// TIA Portal V17 export
// export: Created 2025-04-09T08:02:46.4653844Z, ExportSetting WithDefaults, DisplayName Totally Integrated Automation Portal, DisplayVersion V17 Update 8, DisplayName TIA Portal Openness, DisplayVersion V17 Update 8, DisplayName TIA Portal Version Control Interface, DisplayVersion V17, DisplayName SINAMICS Startdrive Advanced, DisplayVersion V17 SP2, DisplayName SINAMICS Startdrive G110M, G120, G120C, G120D, G120P, G115D, DisplayVersion V17 SP2, DisplayName SINAMICS Startdrive G130, G150, S120, S150, SINAMICS MV, S210, DisplayVersion V17 SP2, DisplayName STEP 7 Professional, DisplayVersion V17 Update 8, DisplayName SINUMERIK ONE STEP 7 Toolbox, DisplayVersion V17 Update 12, DisplayName SINUMERIK ONE PLC Basic Program Plus, DisplayVersion V17 Update 12, DisplayName SINUMERIK 840D sl STEP 7 Toolbox, DisplayVersion V17 Update 12, DisplayName STEP 7 Safety, DisplayVersion V17 Update 6, DisplayName WinCC Advanced, DisplayVersion V17 Update 8
FUNCTION_BLOCK "FB1403_PROGRESSIVE_LUBRICATION_WITH_GREASE"   // FB1403, LAD
{ S7_Optimized_Access := 'FALSE' }
AUTHOR : ETXETAR
VERSION : 1.0
// stored: AutoNumber false, IsIECCheckEnabled false, SetENOAutomatically false, UDAEnableTagReadback false
   VAR_INPUT
      OPTIONS_0 : Byte := 2#0000_0000;   // OPTIONS 0
      OPTIONS_1 : Byte := 2#0000_0000;   // OPTIONS 1
      TIME_VALVE_1 : Time := T#5d;   // H=HOURS; M=MINUTES
      TIME_VALVE_2 : Time := T#5d;   // H=HOURS; M=MINUTES
      TIME_VALVE_3 : Time := T#5d;   // H=HOURS; M=MINUTES
      TIME_VALVE_4 : Time := T#5d;   // H=HOURS; M=MINUTES
      PULSES_PER_CYCLE_VALVE_1 : Int := 2;   // NUMBER OF PULSES PER CYCLE
      PULSES_PER_CYCLE_VALVE_2 : Int := 2;   // NUMBER OF PULSES PER CYCLE
      PULSES_PER_CYCLE_VALVE_3 : Int := 2;   // NUMBER OF PULSES PER CYCLE
      PULSES_PER_CYCLE_VALVE_4 : Int := 2;   // NUMBER OF PULSES PER CYCLE
      BREAKER : Bool;   // CIRCUIT BREAKER INPUT
      LOW_LEVEL_ALM : Bool;   // LOW LEVEL ALARM INPUT
      OVERPRESSURE_ALM : Bool;   // OVERPRESSURE ALARM INPUT
      LUBRICATION_DONE_1 : Bool;   // LUBRICATION_DONE 1 INPUT
      LUBRICATION_DONE_2 : Bool;   // LUBRICATION_DONE 2 INPUT
      LUBRICATION_DONE_3 : Bool;   // LUBRICATION_DONE 3 INPUT
      LUBRICATION_DONE_4 : Bool;   // LUBRICATION_DONE 4 INPUT
      LUBRICATION_DONE_5 : Bool;   // LUBRICATION_DONE 5 INPUT
      LUBRICATION_DONE_6 : Bool;   // LUBRICATION_DONE 6 INPUT
      LUBRICATION_DONE_7 : Bool;   // LUBRICATION_DONE 7 INPUT
      LUBRICATION_DONE_8 : Bool;   // LUBRICATION_DONE 8 INPUT
      LUBRICATION_DONE_9 : Bool;   // LUBRICATION_DONE 9 INPUT
      SWITCH_ON_VALVE_1_DIST_REQ_AXIS_1 : Bool;   // SWITCH ON DISTANCE REQUEST INPUT FOR VALVE 1 AXIS 1
      SWITCH_ON_VALVE_1_DIST_REQ_AXIS_2 : Bool;   // SWITCH ON DISTANCE REQUEST INPUT FOR VALVE 1 AXIS 2
      SWITCH_ON_VALVE_2_DIST_REQ_AXIS_1 : Bool;   // SWITCH ON DISTANCE REQUEST INPUT FOR VALVE 2 AXIS 1
      SWITCH_ON_VALVE_2_DIST_REQ_AXIS_2 : Bool;   // SWITCH ON DISTANCE REQUEST INPUT FOR VALVE 2 AXIS 2
      SWITCH_ON_VALVE_3_DIST_REQ : Bool;   // SWITCH ON DISTANCE REQUEST INPUT FOR VALVE 3
      SWITCH_ON_VALVE_4_DIST_REQ : Bool;   // SWITCH ON DISTANCE REQUEST INPUT FOR VALVE 4
      HMI_REQ_LINE_VALVE_1 : Bool;   // HMI REQUEST LINE
      HMI_REQ_LINE_VALVE_2 : Bool;   // HMI REQUEST LINE
      HMI_REQ_LINE_VALVE_3 : Bool;   // HMI REQUEST LINE
      HMI_REQ_LINE_VALVE_4 : Bool;   // HMI REQUEST LINE
   END_VAR
   VAR_OUTPUT
      HMI_POWER_UP_COND_OFF_VALVE_1 : Bool;   // HMI POWER UP CONDITIONS OFF
      HMI_POWER_UP_COND_ON_VALVE_1 : Bool;   // HMI POWER UP CONDITIONS ON
      HMI_POWER_UP_EXECU_LEFT_VALVE_1 : Bool;   // HMI POWER UP EXECUTABLE LEFT
      HMI_POWER_UP_EXECU_RIGHT_VALVE_1 : Bool;   // HMI POWER UP EXECUTABLE RIGHT
      HMI_POWER_UP_COND_OFF_VALVE_2 : Bool;   // HMI POWER UP CONDITIONS OFF
      HMI_POWER_UP_COND_ON_VALVE_2 : Bool;   // HMI POWER UP CONDITIONS ON
      HMI_POWER_UP_EXECU_LEFT_VALVE_2 : Bool;   // HMI POWER UP EXECUTABLE LEFT
      HMI_POWER_UP_EXECU_RIGHT_VALVE_2 : Bool;   // HMI POWER UP EXECUTABLE RIGHT
      HMI_POWER_UP_COND_OFF_VALVE_3 : Bool;   // HMI POWER UP CONDITIONS OFF
      HMI_POWER_UP_COND_ON_VALVE_3 : Bool;   // HMI POWER UP CONDITIONS ON
      HMI_POWER_UP_EXECU_LEFT_VALVE_3 : Bool;   // HMI POWER UP EXECUTABLE LEFT
      HMI_POWER_UP_EXECU_RIGHT_VALVE_3 : Bool;   // HMI POWER UP EXECUTABLE RIGHT
      HMI_POWER_UP_COND_OFF_VALVE_4 : Bool;   // HMI POWER UP CONDITIONS OFF
      HMI_POWER_UP_COND_ON_VALVE_4 : Bool;   // HMI POWER UP CONDITIONS ON
      HMI_POWER_UP_EXECU_LEFT_VALVE_4 : Bool;   // HMI POWER UP EXECUTABLE LEFT
      HMI_POWER_UP_EXECU_RIGHT_VALVE_4 : Bool;   // HMI POWER UP EXECUTABLE RIGHT
      MOTOR : Bool;   // MOTOR OUTPUT
      VALVE_1 : Bool;
      VALVE_2 : Bool;
      VALVE_3 : Bool;
      VALVE_4 : Bool;
   END_VAR
   VAR DB_SPECIFIC
      BREAKER_ALARM : Bool;   // CIRCUIT BREAKER TRIPPED ALARM
      LOW_LEVEL_ALARM : Bool;   // LOW LEVEL ALARM
      OVERPRESSURE_ALARM : Bool;   // OVERPRESSURE ALARM
      LUBRICATION_DONE_1_ALARM : Bool;   // LUBRICATION DONE 1 ALARM
      LUBRICATION_DONE_2_ALARM : Bool;   // LUBRICATION DONE 2 ALARM
      LUBRICATION_DONE_3_ALARM : Bool;   // LUBRICATION DONE 3 ALARM
      LUBRICATION_DONE_4_ALARM : Bool;   // LUBRICATION DONE 4 ALARM
      DATA_VALVE_1 : Struct
         SWITCH_ON_GENERAL_CONDITIONS : Bool;   // SWITCH ON GENERAL CONDITIONS
         SWITCH_ON_INITIAL_CONDITIONS : Bool;   // SWITCH ON INITIAL CONDITIONS
         SWITCH_ON_MANUAL_REQUEST : Bool;   // SWITCH ON MANUAL REQUEST
         SWITCH_ON_AUTO_REQUEST : Bool;   // SWITCH ON AUTO REQUEST
         SWITCH_ON_TIME_REQUEST : Bool;   // SWITCH ON TIME REQUEST
         SWITCH_ON_GLOBAL_REQUEST : Bool;   // SWITCH ON GLOBAL REQUEST
         SWITCH_ON_CMM : Bool;   // SWITCH ON COMMAND
         SWITCH_ON : Bool;   // SWITCH ON
         IN_SERVICE : Bool;   // IN SERVICE
         SWITCH_OFF_GENERAL_CONDITIONS : Bool;   // SWITCH OFF GENERAL CONDITIONS
         SWITCH_OFF_INITIAL_CONDITIONS : Bool;   // SWITCH OFF INITIAL CONDITIONS
         SWITCH_OFF_MANUAL_REQUEST : Bool;   // SWITCH OFF MANUAL REQUEST
         SWITCH_OFF_AUTO_REQUEST : Bool;   // SWITCH OFF AUTO REQUEST
         SWITCH_OFF_GLOBAL_REQUEST : Bool;   // SWITCH OFF GLOBAL REQUEST
         SWITCH_OFF_CMM : Bool;   // SWITCH OFF COMMAND
         SWITCH_OFF : Bool;   // SWITCH OFF
         OUT_OF_SERVICE : Bool;   // OUT OF SERVICE
         TIMER_1 : TON_TIME;   // TIMER_1
         PULSE_1 : Bool;   // PULSE_1
         PULSE_2 : Bool;   // PULSE_1
      END_STRUCT;
      DATA_VALVE_2 : Struct
         SWITCH_ON_GENERAL_CONDITIONS : Bool;   // SWITCH ON GENERAL CONDITIONS
         SWITCH_ON_INITIAL_CONDITIONS : Bool;   // SWITCH ON INITIAL CONDITIONS
         SWITCH_ON_MANUAL_REQUEST : Bool;   // SWITCH ON MANUAL REQUEST
         SWITCH_ON_AUTO_REQUEST : Bool;   // SWITCH ON AUTO REQUEST
         SWITCH_ON_TIME_REQUEST : Bool;   // SWITCH ON TIME REQUEST
         SWITCH_ON_GLOBAL_REQUEST : Bool;   // SWITCH ON GLOBAL REQUEST
         SWITCH_ON_CMM : Bool;   // SWITCH ON COMMAND
         SWITCH_ON : Bool;   // SWITCH ON
         IN_SERVICE : Bool;   // IN SERVICE
         SWITCH_OFF_GENERAL_CONDITIONS : Bool;   // SWITCH OFF GENERAL CONDITIONS
         SWITCH_OFF_INITIAL_CONDITIONS : Bool;   // SWITCH OFF INITIAL CONDITIONS
         SWITCH_OFF_MANUAL_REQUEST : Bool;   // SWITCH OFF MANUAL REQUEST
         SWITCH_OFF_AUTO_REQUEST : Bool;   // SWITCH OFF AUTO REQUEST
         SWITCH_OFF_GLOBAL_REQUEST : Bool;   // SWITCH OFF GLOBAL REQUEST
         SWITCH_OFF_CMM : Bool;   // SWITCH OFF COMMAND
         SWITCH_OFF : Bool;   // SWITCH OFF
         OUT_OF_SERVICE : Bool;   // OUT OF SERVICE
         TIMER_1 : TON_TIME;   // TIMER_1
         PULSE_1 : Bool;   // PULSE_1
         PULSE_2 : Bool;   // PULSE_1
      END_STRUCT;
      DATA_VALVE_3 : Struct
         SWITCH_ON_GENERAL_CONDITIONS : Bool;   // SWITCH ON GENERAL CONDITIONS
         SWITCH_ON_INITIAL_CONDITIONS : Bool;   // SWITCH ON INITIAL CONDITIONS
         SWITCH_ON_MANUAL_REQUEST : Bool;   // SWITCH ON MANUAL REQUEST
         SWITCH_ON_AUTO_REQUEST : Bool;   // SWITCH ON AUTO REQUEST
         SWITCH_ON_TIME_REQUEST : Bool;   // SWITCH ON TIME REQUEST
         SWITCH_ON_GLOBAL_REQUEST : Bool;   // SWITCH ON GLOBAL REQUEST
         SWITCH_ON_CMM : Bool;   // SWITCH ON COMMAND
         SWITCH_ON : Bool;   // SWITCH ON
         IN_SERVICE : Bool;   // IN SERVICE
         SWITCH_OFF_GENERAL_CONDITIONS : Bool;   // SWITCH OFF GENERAL CONDITIONS
         SWITCH_OFF_INITIAL_CONDITIONS : Bool;   // SWITCH OFF INITIAL CONDITIONS
         SWITCH_OFF_MANUAL_REQUEST : Bool;   // SWITCH OFF MANUAL REQUEST
         SWITCH_OFF_AUTO_REQUEST : Bool;   // SWITCH OFF AUTO REQUEST
         SWITCH_OFF_GLOBAL_REQUEST : Bool;   // SWITCH OFF GLOBAL REQUEST
         SWITCH_OFF_CMM : Bool;   // SWITCH OFF COMMAND
         SWITCH_OFF : Bool;   // SWITCH OFF
         OUT_OF_SERVICE : Bool;   // OUT OF SERVICE
         TIMER_1 : TON_TIME;   // TIMER_1
         PULSE_1 : Bool;   // PULSE_1
         PULSE_2 : Bool;   // PULSE_1
      END_STRUCT;
      DATA_VALVE_4 : Struct
         SWITCH_ON_GENERAL_CONDITIONS : Bool;   // SWITCH ON GENERAL CONDITIONS
         SWITCH_ON_INITIAL_CONDITIONS : Bool;   // SWITCH ON INITIAL CONDITIONS
         SWITCH_ON_MANUAL_REQUEST : Bool;   // SWITCH ON MANUAL REQUEST
         SWITCH_ON_AUTO_REQUEST : Bool;   // SWITCH ON AUTO REQUEST
         SWITCH_ON_TIME_REQUEST : Bool;   // SWITCH ON TIME REQUEST
         SWITCH_ON_GLOBAL_REQUEST : Bool;   // SWITCH ON GLOBAL REQUEST
         SWITCH_ON_CMM : Bool;   // SWITCH ON COMMAND
         SWITCH_ON : Bool;   // SWITCH ON
         IN_SERVICE : Bool;   // IN SERVICE
         SWITCH_OFF_GENERAL_CONDITIONS : Bool;   // SWITCH OFF GENERAL CONDITIONS
         SWITCH_OFF_INITIAL_CONDITIONS : Bool;   // SWITCH OFF INITIAL CONDITIONS
         SWITCH_OFF_MANUAL_REQUEST : Bool;   // SWITCH OFF MANUAL REQUEST
         SWITCH_OFF_AUTO_REQUEST : Bool;   // SWITCH OFF AUTO REQUEST
         SWITCH_OFF_GLOBAL_REQUEST : Bool;   // SWITCH OFF GLOBAL REQUEST
         SWITCH_OFF_CMM : Bool;   // SWITCH OFF COMMAND
         SWITCH_OFF : Bool;   // SWITCH OFF
         OUT_OF_SERVICE : Bool;   // OUT OF SERVICE
         TIMER_1 : TON_TIME;   // TIMER_1
         PULSE_1 : Bool;   // PULSE_1
         PULSE_2 : Bool;   // PULSE_1
      END_STRUCT;
      CYCLE_IN_PROCESS : Bool;   // CYCLE IN PROCESS
      ALL_LUBRICATION_DONE : Bool;   // ALL LUBRICATION DONE
      ALL_LUBRICATION_DONE_DELAYED : Bool;   // ALL LUBRICATION DONE DELAYED
      SWITCH_ON_MOTOR_REQUEST : Bool;   // SWITCH ON MOTOR REQUEST
      ANY_CYCLE_NOT_DONE : Bool;   // ANY CYCLE NOT DONE
      CYCLE_FINISHED_1 : Bool;   // CYCLE FINISHED 1
      CYCLE_FINISHED_2 : Bool;   // CYCLE FINISHED 2
      CYCLE_FINISHED_3 : Bool;   // CYCLE FINISHED 3
      CYCLE_FINISHED_4 : Bool;   // CYCLE FINISHED 4
      MANUAL_REQUEST_HELP : Bool;   // MANUAL REQUEST HELP
      SWITCH_ON_GENERAL_CONDITION_HELP : Bool;   // SWITCH ON GENERAL CONDITION HELP
      SWITCH_ON_INITIAL_CONDITION_HELP : Bool;   // SWITCH ON INITIAL CONDITION HELP
      SWITCH_OFF_GENERAL_CONDITION_HELP : Bool;   // SWITCH OFF GENERAL CONDITION HELP
      SWITCH_OFF_INITIAL_CONDITION_HELP : Bool;   // SWITCH OFF INITIAL CONDITION HELP
      ANY_ACTIVE_ALARM : Bool;   // ANY ACTIVE ALARM
      SEOC_ALARMS : Bool;   // STOP END OF CYCLE ALARMS
      WARNINGS : Bool;   // WARNINGS
      WARNINGS_GONE : Bool;   // WARNINGS GONE
      TIMER_AUX_SWTICH_ON_MOTOR : TON_TIME;   // SWTICH ON MOTOR TIMER
      TIMER_ALL_LUBRICATION_DONE : TON_TIME;   // ALL LUBRICATION DONE TIMER
      TIMER_LOW_LEVEL_ALM : TON_TIME;   // LOW LEVEL TIMER
      TIMER_OVERPRESSURE_ALM : TON_TIME;   // OVERPRESSURE TIMER
      TIMER_ANY_CYCLE_NOT_DONE : TON_TIME;   // ANY CYCLE NOT DONE TIMER
      TIMER_RUN_NIGHT_TEST : TON_TIME;   // TIMER RUN NIGHT TEST
      COUNTER_1 { S7_SetPoint := 'True'} : CTU_INT;
      COUNTER_2 { S7_SetPoint := 'True'} : CTU_INT;
      COUNTER_3 { S7_SetPoint := 'True'} : CTU_INT;
      COUNTER_4 { S7_SetPoint := 'True'} : CTU_INT;
      SEQ_GLOBAL_AUTO_REQ : Bool;   // SEQUENCE GLOBAL AUTO REQUEST
      PULSE_1 : Bool;
      PULSE_2 : Bool;
      PULSE_3 : Bool;
      PULSE_4 : Bool;
      PULSE_5 : Bool;
      PULSE_6 : Bool;
      PULSE_7 : Bool;
      PULSE_8 : Bool;
      VALVE_1_AXIS_1_DIST_MEM_REQ : Bool;   // VALVE 1 AXIS 1 DISTANCE MEMORY REQUEST
      VALVE_1_AXIS_2_DIST_MEM_REQ : Bool;   // VALVE 1 AXIS 2 DISTANCE MEMORY REQUEST
      VALVE_2_AXIS_1_DIST_MEM_REQ : Bool;   // VALVE 2 AXIS 1 DISTANCE MEMORY REQUEST
      VALVE_2_AXIS_2_DIST_MEM_REQ : Bool;   // VALVE 2 AXIS 2 DISTANCE MEMORY REQUEST
      VALVE_1_AXIS_1_2_DIST_REQ : Bool;   // VALVE 1 AXIS 1 & 2 DISTANCE REQUEST
      VALVE_2_AXIS_1_2_DIST_REQ : Bool;   // VALVE 2 AXIS 1 & 2 DISTANCE REQUEST
   END_VAR
   VAR_TEMP
      INPUTS_MASK : Byte;   // INPUT MASK
      O_BYTE_0 : Struct   // OPTIONS BYTE 0
         "CIRCUIT BREAKER" : Bool;   // CIRCUIT BREAKER OPTION
         LOW_LEVEL_ALARM : Bool;   // LOW LEVEL ALARM OPTION
         OVERPRESSURE_ALARM : Bool;   // OVERPRESSURE ALARM OPTION
         LUBRICATION_BY_TIME_VALVE_1 : Bool;   // LUBRICATE BY TIMER OR BY AUTO REQUEST OPTION
         LUBRICATION_BY_TIME_VALVE_2 : Bool;   // LUBRICATE BY TIMER OR BY AUTO REQUEST OPTION
         LUBRICATION_BY_TIME_VALVE_3 : Bool;   // LUBRICATE BY TIMER OR BY AUTO REQUEST OPTION
         LUBRICATION_BY_TIME_VALVE_4 : Bool;   // LUBRICATE BY TIMER OR BY AUTO REQUEST OPTION
         LUBRICATION_DONE_1 : Bool;   // LUBRICATION DONE 1 OPTION
      END_STRUCT;
      O_BYTE_1 : Struct   // OPTIONS BYTE 0
         LUBRICATION_DONE_2 : Bool;   // LUBRICATION DONE 2 OPTION
         LUBRICATION_DONE_3 : Bool;   // LUBRICATION DONE 2 OPTION
         LUBRICATION_DONE_4 : Bool;   // LUBRICATION DONE 2 OPTION
         LUBRICATION_DONE_5 : Bool;   // LUBRICATION DONE 2 OPTION
         LUBRICATION_DONE_6 : Bool;   // LUBRICATION DONE 2 OPTION
         LUBRICATION_DONE_7 : Bool;   // LUBRICATION DONE 2 OPTION
         LUBRICATION_DONE_8 : Bool;   // LUBRICATION DONE 2 OPTION
         LUBRICATION_DONE_9 : Bool;   // LUBRICATION DONE 2 OPTION
      END_STRUCT;
      DB_NUMBER : DInt;   // DB NUMBER FOR ALARM AND HELP DECODING
   END_VAR
   // TIMER_AUX_SWTICH_ON_MOTOR.PT := T#2h;
   // TIMER_ALL_LUBRICATION_DONE.PT := T#1s;
   // TIMER_LOW_LEVEL_ALM.PT := T#5s;
   // TIMER_OVERPRESSURE_ALM.PT := T#5s;
   // TIMER_ANY_CYCLE_NOT_DONE.PT := T#11M;
   // TIMER_RUN_NIGHT_TEST.PT := T#10M;
   VAR_TEMP   // added for the SCL form of the ladder/FBD networks
      _w1 : Bool;
      _w2 : Bool;
      _w3 : Bool;
      _w4 : Bool;
      _w5 : Bool;
      _w6 : Bool;
      _w7 : Bool;
      _w8 : Bool;
   END_VAR
BEGIN

NETWORK
TITLE = READ INSTANCE DB
      L     DINO;
      +     10#800000;
      T     #DB_NUMBER;


REGION Network 2: OPTIONS
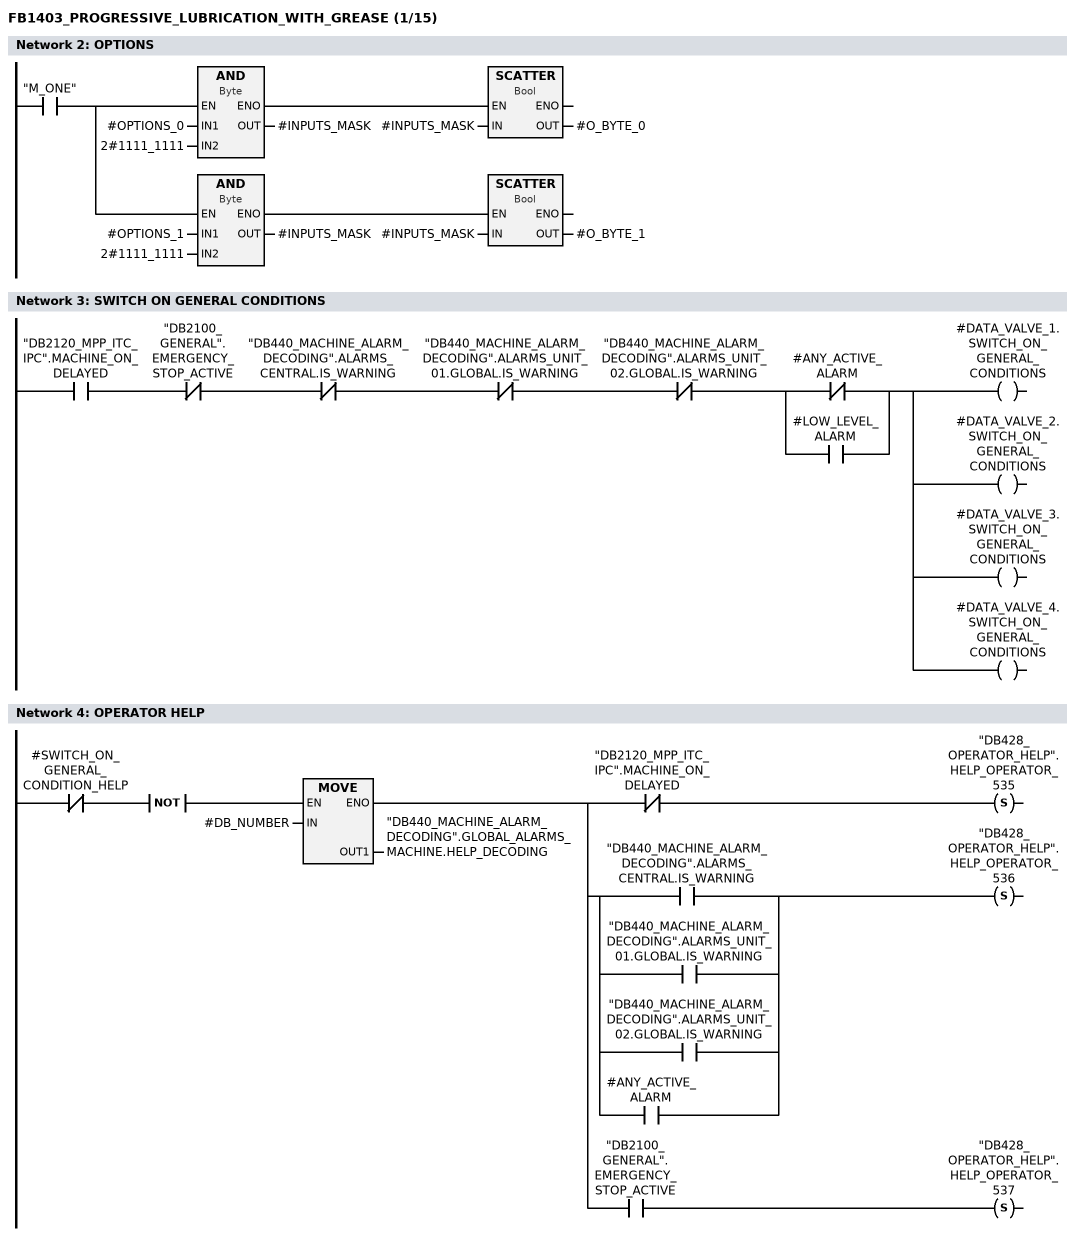
   RUNG wire#powerrail
      Contact( "M_ONE" )
      wire#w1
      { S7_Templates := "SrcType := Byte"; S7_GenerateENO := "TRUE" } And(in1 := #OPTIONS_0, in2 := 2#1111_1111, out => #INPUTS_MASK)
      { S7_Templates := "[dest_type := Bool, src_type := Byte]" } SCATTER(IN := #INPUTS_MASK, OUT => #O_BYTE_0)
   END_RUNG
   RUNG wire#w1
      { S7_Templates := "SrcType := Byte"; S7_GenerateENO := "TRUE" } And(in1 := #OPTIONS_1, in2 := 2#1111_1111, out => #INPUTS_MASK)
      { S7_Templates := "[dest_type := Bool, src_type := Byte]" } SCATTER(IN := #INPUTS_MASK, OUT => #O_BYTE_1)
   END_RUNG
   // the same network as SCL:
   IF "M_ONE" THEN #INPUTS_MASK := #OPTIONS_0 AND 2#1111_1111; END_IF;
   #_w1 := "M_ONE";
   IF #_w1 THEN
       SCATTER(IN := #INPUTS_MASK, OUT => #O_BYTE_0);
       #INPUTS_MASK := #OPTIONS_1 AND 2#1111_1111;
       SCATTER(IN := #INPUTS_MASK, OUT => #O_BYTE_1);
   END_IF;
END_REGION

REGION Network 3: SWITCH ON GENERAL CONDITIONS
   RUNG wire#powerrail
      Contact( "DB2120_MPP_ITC_IPC".MACHINE_ON_DELAYED )
      I_Contact( "DB2100_GENERAL".EMERGENCY_STOP_ACTIVE )
      I_Contact( "DB440_MACHINE_ALARM_DECODING".ALARMS_CENTRAL.IS_WARNING )
      I_Contact( "DB440_MACHINE_ALARM_DECODING".ALARMS_UNIT_01.GLOBAL.IS_WARNING )
      I_Contact( "DB440_MACHINE_ALARM_DECODING".ALARMS_UNIT_02.GLOBAL.IS_WARNING )
      wire#w1
      I_Contact( #ANY_ACTIVE_ALARM )
      wire#w2
      Coil( #DATA_VALVE_1.SWITCH_ON_GENERAL_CONDITIONS )
   END_RUNG
   RUNG wire#w1
      Contact( #LOW_LEVEL_ALARM )
   END_RUNG wire#w2
   RUNG wire#w2
      Coil( #DATA_VALVE_2.SWITCH_ON_GENERAL_CONDITIONS )
   END_RUNG
   RUNG wire#w2
      Coil( #DATA_VALVE_3.SWITCH_ON_GENERAL_CONDITIONS )
   END_RUNG
   RUNG wire#w2
      Coil( #DATA_VALVE_4.SWITCH_ON_GENERAL_CONDITIONS )
   END_RUNG
   // the same network as SCL:
   #DATA_VALVE_1.SWITCH_ON_GENERAL_CONDITIONS := "DB2120_MPP_ITC_IPC".MACHINE_ON_DELAYED AND NOT "DB2100_GENERAL".EMERGENCY_STOP_ACTIVE AND NOT "DB440_MACHINE_ALARM_DECODING".ALARMS_CENTRAL.IS_WARNING AND NOT "DB440_MACHINE_ALARM_DECODING".ALARMS_UNIT_01.GLOBAL.IS_WARNING AND NOT "DB440_MACHINE_ALARM_DECODING".ALARMS_UNIT_02.GLOBAL.IS_WARNING AND (NOT #ANY_ACTIVE_ALARM OR #LOW_LEVEL_ALARM);
   #DATA_VALVE_2.SWITCH_ON_GENERAL_CONDITIONS := #DATA_VALVE_1.SWITCH_ON_GENERAL_CONDITIONS;
   #DATA_VALVE_3.SWITCH_ON_GENERAL_CONDITIONS := #DATA_VALVE_1.SWITCH_ON_GENERAL_CONDITIONS;
   #DATA_VALVE_4.SWITCH_ON_GENERAL_CONDITIONS := #DATA_VALVE_1.SWITCH_ON_GENERAL_CONDITIONS;
END_REGION

REGION Network 4: OPERATOR HELP
   RUNG wire#powerrail
      I_Contact( #SWITCH_ON_GENERAL_CONDITION_HELP )
      Not()
      { S7_GenerateENO := "TRUE" } Move(in := #DB_NUMBER, out1 => "DB440_MACHINE_ALARM_DECODING".GLOBAL_ALARMS_MACHINE.HELP_DECODING)
      wire#w1
      I_Contact( "DB2120_MPP_ITC_IPC".MACHINE_ON_DELAYED )
      S_Coil( "DB428_OPERATOR_HELP".HELP_OPERATOR_535 )
   END_RUNG
   RUNG wire#w1
      Contact( "DB440_MACHINE_ALARM_DECODING".ALARMS_CENTRAL.IS_WARNING )
      wire#w2
      S_Coil( "DB428_OPERATOR_HELP".HELP_OPERATOR_536 )
   END_RUNG
   RUNG wire#w1
      Contact( "DB440_MACHINE_ALARM_DECODING".ALARMS_UNIT_01.GLOBAL.IS_WARNING )
   END_RUNG wire#w2
   RUNG wire#w1
      Contact( "DB440_MACHINE_ALARM_DECODING".ALARMS_UNIT_02.GLOBAL.IS_WARNING )
   END_RUNG wire#w2
   RUNG wire#w1
      Contact( #ANY_ACTIVE_ALARM )
   END_RUNG wire#w2
   RUNG wire#w1
      Contact( "DB2100_GENERAL".EMERGENCY_STOP_ACTIVE )
      S_Coil( "DB428_OPERATOR_HELP".HELP_OPERATOR_537 )
   END_RUNG
   // the same network as SCL:
   // ENO of a box is taken as its EN; it also drops when the box reports an error
   #_w1 := NOT (NOT #SWITCH_ON_GENERAL_CONDITION_HELP);
   IF #_w1 THEN "DB440_MACHINE_ALARM_DECODING".GLOBAL_ALARMS_MACHINE.HELP_DECODING := #DB_NUMBER; END_IF;
   IF #_w1 AND NOT "DB2120_MPP_ITC_IPC".MACHINE_ON_DELAYED THEN
       "DB428_OPERATOR_HELP".HELP_OPERATOR_535 := TRUE;
   END_IF;
   IF #_w1 AND ("DB440_MACHINE_ALARM_DECODING".ALARMS_CENTRAL.IS_WARNING OR "DB440_MACHINE_ALARM_DECODING".ALARMS_UNIT_01.GLOBAL.IS_WARNING OR "DB440_MACHINE_ALARM_DECODING".ALARMS_UNIT_02.GLOBAL.IS_WARNING OR #ANY_ACTIVE_ALARM) THEN
       "DB428_OPERATOR_HELP".HELP_OPERATOR_536 := TRUE;
   END_IF;
   IF #_w1 AND "DB2100_GENERAL".EMERGENCY_STOP_ACTIVE THEN
       "DB428_OPERATOR_HELP".HELP_OPERATOR_537 := TRUE;
   END_IF;
END_REGION

REGION Network 5: SWITCH ON INITIAL CONDITIONS
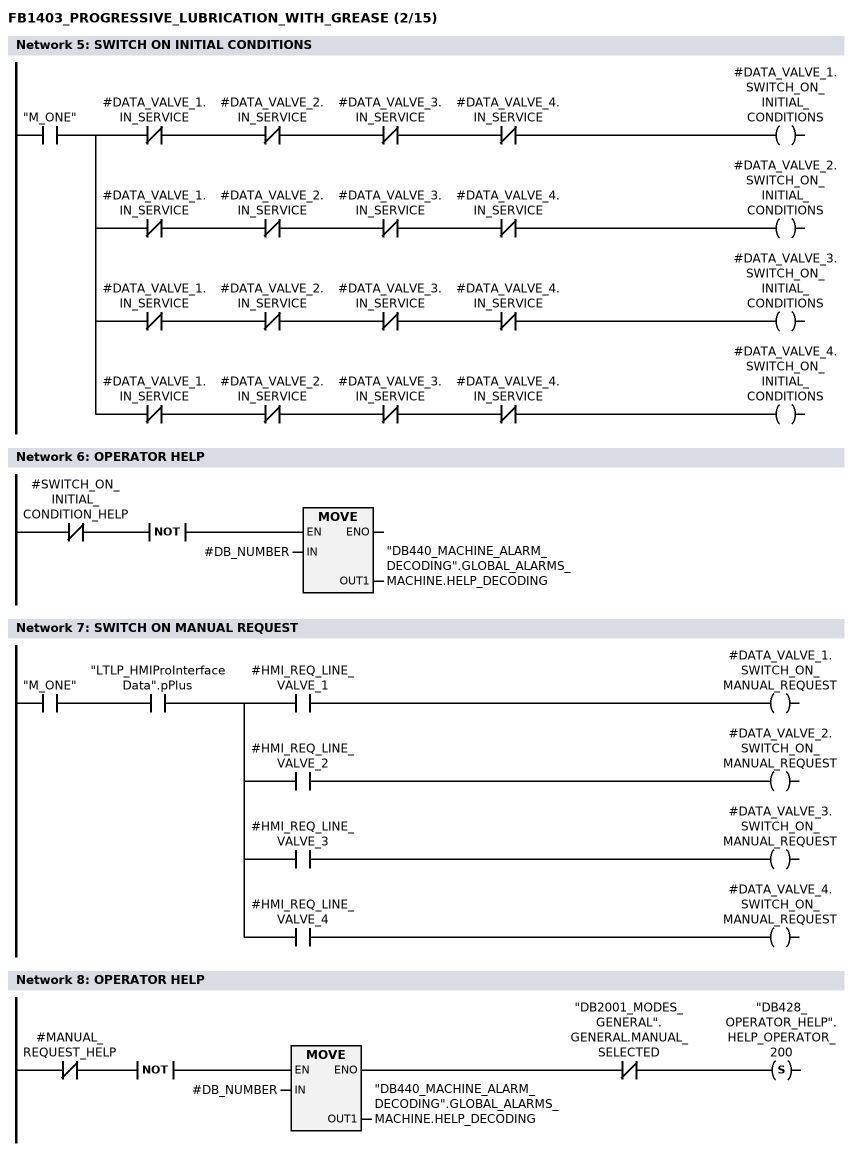
   RUNG wire#powerrail
      Contact( "M_ONE" )
      wire#w1
      I_Contact( #DATA_VALVE_1.IN_SERVICE )
      I_Contact( #DATA_VALVE_2.IN_SERVICE )
      I_Contact( #DATA_VALVE_3.IN_SERVICE )
      I_Contact( #DATA_VALVE_4.IN_SERVICE )
      Coil( #DATA_VALVE_1.SWITCH_ON_INITIAL_CONDITIONS )
   END_RUNG
   RUNG wire#w1
      I_Contact( #DATA_VALVE_1.IN_SERVICE )
      I_Contact( #DATA_VALVE_2.IN_SERVICE )
      I_Contact( #DATA_VALVE_3.IN_SERVICE )
      I_Contact( #DATA_VALVE_4.IN_SERVICE )
      Coil( #DATA_VALVE_2.SWITCH_ON_INITIAL_CONDITIONS )
   END_RUNG
   RUNG wire#w1
      I_Contact( #DATA_VALVE_1.IN_SERVICE )
      I_Contact( #DATA_VALVE_2.IN_SERVICE )
      I_Contact( #DATA_VALVE_3.IN_SERVICE )
      I_Contact( #DATA_VALVE_4.IN_SERVICE )
      Coil( #DATA_VALVE_3.SWITCH_ON_INITIAL_CONDITIONS )
   END_RUNG
   RUNG wire#w1
      I_Contact( #DATA_VALVE_1.IN_SERVICE )
      I_Contact( #DATA_VALVE_2.IN_SERVICE )
      I_Contact( #DATA_VALVE_3.IN_SERVICE )
      I_Contact( #DATA_VALVE_4.IN_SERVICE )
      Coil( #DATA_VALVE_4.SWITCH_ON_INITIAL_CONDITIONS )
   END_RUNG
   // the same network as SCL:
   #DATA_VALVE_1.SWITCH_ON_INITIAL_CONDITIONS := "M_ONE" AND NOT #DATA_VALVE_1.IN_SERVICE AND NOT #DATA_VALVE_2.IN_SERVICE AND NOT #DATA_VALVE_3.IN_SERVICE AND NOT #DATA_VALVE_4.IN_SERVICE;
   #DATA_VALVE_2.SWITCH_ON_INITIAL_CONDITIONS := "M_ONE" AND NOT #DATA_VALVE_1.IN_SERVICE AND NOT #DATA_VALVE_2.IN_SERVICE AND NOT #DATA_VALVE_3.IN_SERVICE AND NOT #DATA_VALVE_4.IN_SERVICE;
   #DATA_VALVE_3.SWITCH_ON_INITIAL_CONDITIONS := "M_ONE" AND NOT #DATA_VALVE_1.IN_SERVICE AND NOT #DATA_VALVE_2.IN_SERVICE AND NOT #DATA_VALVE_3.IN_SERVICE AND NOT #DATA_VALVE_4.IN_SERVICE;
   #DATA_VALVE_4.SWITCH_ON_INITIAL_CONDITIONS := "M_ONE" AND NOT #DATA_VALVE_1.IN_SERVICE AND NOT #DATA_VALVE_2.IN_SERVICE AND NOT #DATA_VALVE_3.IN_SERVICE AND NOT #DATA_VALVE_4.IN_SERVICE;
END_REGION

REGION Network 6: OPERATOR HELP
   RUNG wire#powerrail
      I_Contact( #SWITCH_ON_INITIAL_CONDITION_HELP )
      Not()
      { S7_GenerateENO := "TRUE" } Move(in := #DB_NUMBER, out1 => "DB440_MACHINE_ALARM_DECODING".GLOBAL_ALARMS_MACHINE.HELP_DECODING)
   END_RUNG
   // the same network as SCL:
   IF NOT (NOT #SWITCH_ON_INITIAL_CONDITION_HELP) THEN
       "DB440_MACHINE_ALARM_DECODING".GLOBAL_ALARMS_MACHINE.HELP_DECODING := #DB_NUMBER;
   END_IF;
END_REGION

REGION Network 7: SWITCH ON MANUAL REQUEST
   RUNG wire#powerrail
      Contact( "M_ONE" )
      Contact( "LTLP_HMIProInterfaceData".pPlus )
      wire#w1
      Contact( #HMI_REQ_LINE_VALVE_1 )
      Coil( #DATA_VALVE_1.SWITCH_ON_MANUAL_REQUEST )
   END_RUNG
   RUNG wire#w1
      Contact( #HMI_REQ_LINE_VALVE_2 )
      Coil( #DATA_VALVE_2.SWITCH_ON_MANUAL_REQUEST )
   END_RUNG
   RUNG wire#w1
      Contact( #HMI_REQ_LINE_VALVE_3 )
      Coil( #DATA_VALVE_3.SWITCH_ON_MANUAL_REQUEST )
   END_RUNG
   RUNG wire#w1
      Contact( #HMI_REQ_LINE_VALVE_4 )
      Coil( #DATA_VALVE_4.SWITCH_ON_MANUAL_REQUEST )
   END_RUNG
   // the same network as SCL:
   #_w1 := "M_ONE" AND "LTLP_HMIProInterfaceData".pPlus;
   #DATA_VALVE_1.SWITCH_ON_MANUAL_REQUEST := #_w1 AND #HMI_REQ_LINE_VALVE_1;
   #DATA_VALVE_2.SWITCH_ON_MANUAL_REQUEST := #_w1 AND #HMI_REQ_LINE_VALVE_2;
   #DATA_VALVE_3.SWITCH_ON_MANUAL_REQUEST := #_w1 AND #HMI_REQ_LINE_VALVE_3;
   #DATA_VALVE_4.SWITCH_ON_MANUAL_REQUEST := #_w1 AND #HMI_REQ_LINE_VALVE_4;
END_REGION

REGION Network 8: OPERATOR HELP
   RUNG wire#powerrail
      I_Contact( #MANUAL_REQUEST_HELP )
      Not()
      { S7_GenerateENO := "TRUE" } Move(in := #DB_NUMBER, out1 => "DB440_MACHINE_ALARM_DECODING".GLOBAL_ALARMS_MACHINE.HELP_DECODING)
      I_Contact( "DB2001_MODES_GENERAL".GENERAL.MANUAL_SELECTED )
      S_Coil( "DB428_OPERATOR_HELP".HELP_OPERATOR_200 )
   END_RUNG
   // the same network as SCL:
   // ENO of a box is taken as its EN; it also drops when the box reports an error
   #_w1 := NOT (NOT #MANUAL_REQUEST_HELP);
   IF #_w1 THEN "DB440_MACHINE_ALARM_DECODING".GLOBAL_ALARMS_MACHINE.HELP_DECODING := #DB_NUMBER; END_IF;
   IF #_w1 AND NOT "DB2001_MODES_GENERAL".GENERAL.MANUAL_SELECTED THEN
       "DB428_OPERATOR_HELP".HELP_OPERATOR_200 := TRUE;
   END_IF;
END_REGION

REGION Network 9: SWITCH ON DISTANCE REQUEST ACTIVATION WITH 2 AXIS
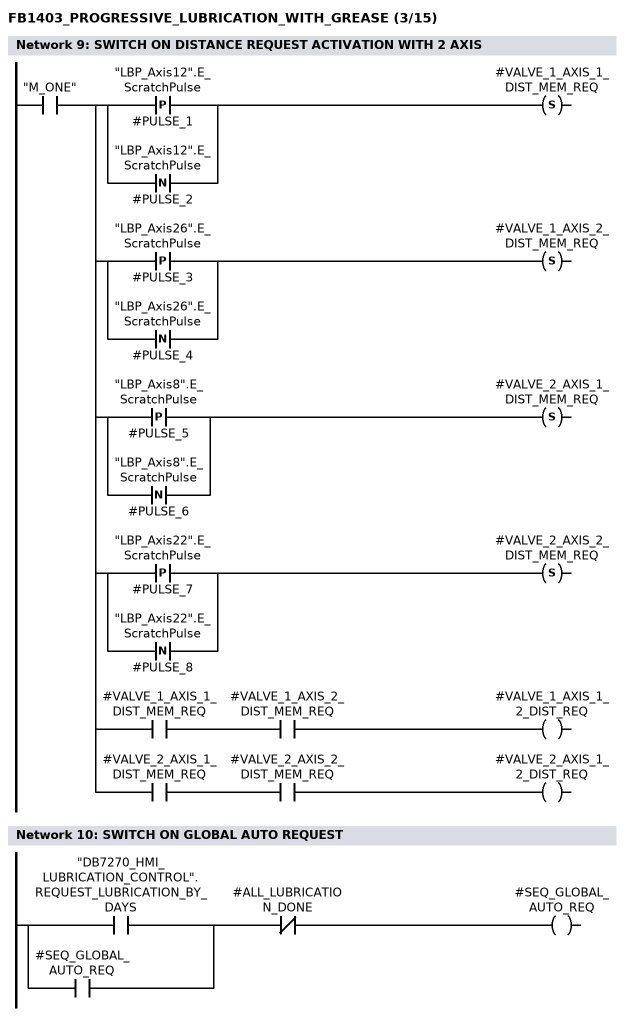
   RUNG wire#powerrail
      Contact( "M_ONE" )
      wire#w1
      P_Contact(operand := "LBP_Axis12".E_ScratchPulse, bit := #PULSE_1)
      wire#w2
      S_Coil( #VALVE_1_AXIS_1_DIST_MEM_REQ )
   END_RUNG
   RUNG wire#w1
      N_Contact(operand := "LBP_Axis12".E_ScratchPulse, bit := #PULSE_2)
   END_RUNG wire#w2
   RUNG wire#w1
      P_Contact(operand := "LBP_Axis26".E_ScratchPulse, bit := #PULSE_3)
      wire#w3
      S_Coil( #VALVE_1_AXIS_2_DIST_MEM_REQ )
   END_RUNG
   RUNG wire#w1
      N_Contact(operand := "LBP_Axis26".E_ScratchPulse, bit := #PULSE_4)
   END_RUNG wire#w3
   RUNG wire#w1
      P_Contact(operand := "LBP_Axis8".E_ScratchPulse, bit := #PULSE_5)
      wire#w4
      S_Coil( #VALVE_2_AXIS_1_DIST_MEM_REQ )
   END_RUNG
   RUNG wire#w1
      N_Contact(operand := "LBP_Axis8".E_ScratchPulse, bit := #PULSE_6)
   END_RUNG wire#w4
   RUNG wire#w1
      P_Contact(operand := "LBP_Axis22".E_ScratchPulse, bit := #PULSE_7)
      wire#w5
      S_Coil( #VALVE_2_AXIS_2_DIST_MEM_REQ )
   END_RUNG
   RUNG wire#w1
      N_Contact(operand := "LBP_Axis22".E_ScratchPulse, bit := #PULSE_8)
   END_RUNG wire#w5
   RUNG wire#w1
      Contact( #VALVE_1_AXIS_1_DIST_MEM_REQ )
      Contact( #VALVE_1_AXIS_2_DIST_MEM_REQ )
      Coil( #VALVE_1_AXIS_1_2_DIST_REQ )
   END_RUNG
   RUNG wire#w1
      Contact( #VALVE_2_AXIS_1_DIST_MEM_REQ )
      Contact( #VALVE_2_AXIS_2_DIST_MEM_REQ )
      Coil( #VALVE_2_AXIS_1_2_DIST_REQ )
   END_RUNG
   // the same network as SCL:
   #_w1 := "M_ONE" AND "LBP_Axis12".E_ScratchPulse AND NOT #PULSE_1;   // rising edge of "LBP_Axis12".E_ScratchPulse
   #PULSE_1 := "LBP_Axis12".E_ScratchPulse;
   #_w2 := "M_ONE" AND NOT "LBP_Axis12".E_ScratchPulse AND #PULSE_2;   // falling edge of "LBP_Axis12".E_ScratchPulse
   #PULSE_2 := "LBP_Axis12".E_ScratchPulse;
   IF #_w1 OR #_w2 THEN #VALVE_1_AXIS_1_DIST_MEM_REQ := TRUE; END_IF;
   #_w3 := "M_ONE" AND "LBP_Axis26".E_ScratchPulse AND NOT #PULSE_3;   // rising edge of "LBP_Axis26".E_ScratchPulse
   #PULSE_3 := "LBP_Axis26".E_ScratchPulse;
   #_w4 := "M_ONE" AND NOT "LBP_Axis26".E_ScratchPulse AND #PULSE_4;   // falling edge of "LBP_Axis26".E_ScratchPulse
   #PULSE_4 := "LBP_Axis26".E_ScratchPulse;
   IF #_w3 OR #_w4 THEN #VALVE_1_AXIS_2_DIST_MEM_REQ := TRUE; END_IF;
   #_w5 := "M_ONE" AND "LBP_Axis8".E_ScratchPulse AND NOT #PULSE_5;   // rising edge of "LBP_Axis8".E_ScratchPulse
   #PULSE_5 := "LBP_Axis8".E_ScratchPulse;
   #_w6 := "M_ONE" AND NOT "LBP_Axis8".E_ScratchPulse AND #PULSE_6;   // falling edge of "LBP_Axis8".E_ScratchPulse
   #PULSE_6 := "LBP_Axis8".E_ScratchPulse;
   IF #_w5 OR #_w6 THEN #VALVE_2_AXIS_1_DIST_MEM_REQ := TRUE; END_IF;
   #_w7 := "M_ONE" AND "LBP_Axis22".E_ScratchPulse AND NOT #PULSE_7;   // rising edge of "LBP_Axis22".E_ScratchPulse
   #PULSE_7 := "LBP_Axis22".E_ScratchPulse;
   #_w8 := "M_ONE" AND NOT "LBP_Axis22".E_ScratchPulse AND #PULSE_8;   // falling edge of "LBP_Axis22".E_ScratchPulse
   #PULSE_8 := "LBP_Axis22".E_ScratchPulse;
   IF #_w7 OR #_w8 THEN #VALVE_2_AXIS_2_DIST_MEM_REQ := TRUE; END_IF;
   #VALVE_1_AXIS_1_2_DIST_REQ := "M_ONE" AND #VALVE_1_AXIS_1_DIST_MEM_REQ AND #VALVE_1_AXIS_2_DIST_MEM_REQ;
   #VALVE_2_AXIS_1_2_DIST_REQ := "M_ONE" AND #VALVE_2_AXIS_1_DIST_MEM_REQ AND #VALVE_2_AXIS_2_DIST_MEM_REQ;
END_REGION

REGION Network 10: SWITCH ON GLOBAL AUTO REQUEST
   RUNG wire#powerrail
      Contact( "DB7270_HMI_LUBRICATION_CONTROL".REQUEST_LUBRICATION_BY_DAYS )
      wire#w1
      I_Contact( #ALL_LUBRICATION_DONE )
      Coil( #SEQ_GLOBAL_AUTO_REQ )
   END_RUNG
   RUNG wire#powerrail
      Contact( #SEQ_GLOBAL_AUTO_REQ )
   END_RUNG wire#w1
   // the same network as SCL:
   #SEQ_GLOBAL_AUTO_REQ := ("DB7270_HMI_LUBRICATION_CONTROL".REQUEST_LUBRICATION_BY_DAYS OR #SEQ_GLOBAL_AUTO_REQ) AND NOT #ALL_LUBRICATION_DONE;
END_REGION

REGION Network 11: SWITCH ON AUTO REQUEST (DISTANCE SPECIFIC OR FIRST SCAN (ALL))
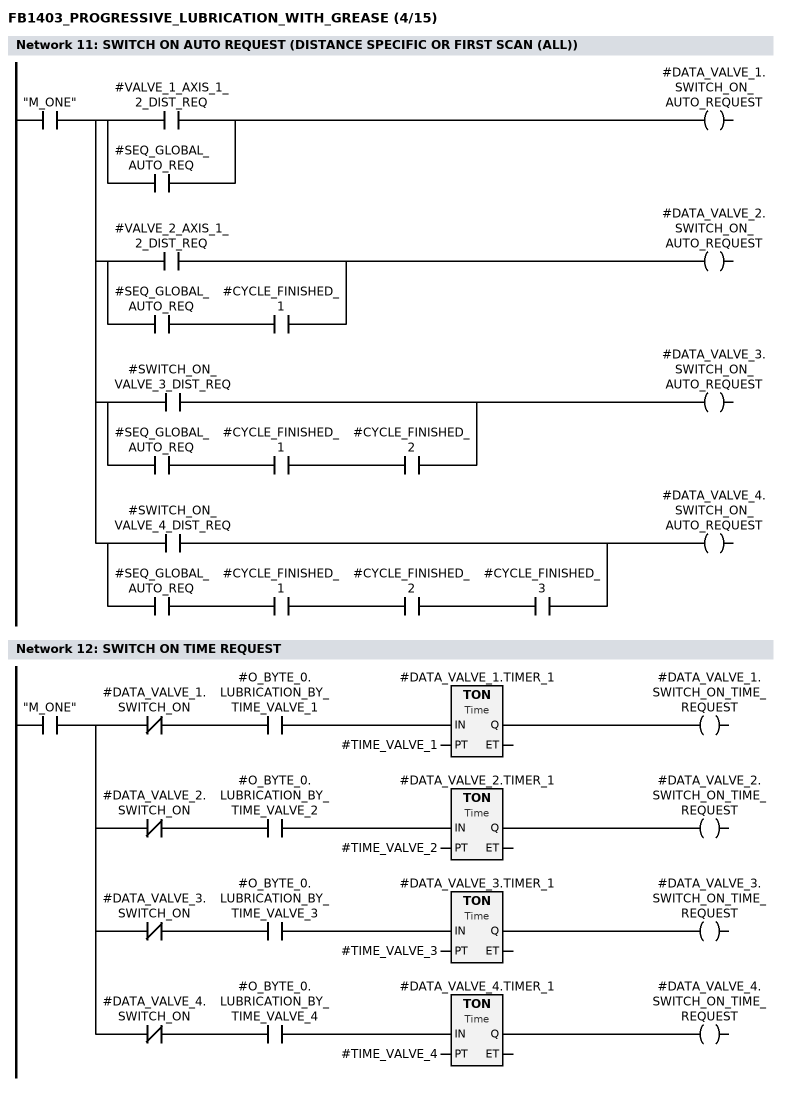
   RUNG wire#powerrail
      Contact( "M_ONE" )
      wire#w1
      Contact( #VALVE_1_AXIS_1_2_DIST_REQ )
      wire#w2
      Coil( #DATA_VALVE_1.SWITCH_ON_AUTO_REQUEST )
   END_RUNG
   RUNG wire#w1
      Contact( #SEQ_GLOBAL_AUTO_REQ )
   END_RUNG wire#w2
   RUNG wire#w1
      Contact( #VALVE_2_AXIS_1_2_DIST_REQ )
      wire#w3
      Coil( #DATA_VALVE_2.SWITCH_ON_AUTO_REQUEST )
   END_RUNG
   RUNG wire#w1
      Contact( #SEQ_GLOBAL_AUTO_REQ )
      Contact( #CYCLE_FINISHED_1 )
   END_RUNG wire#w3
   RUNG wire#w1
      Contact( #SWITCH_ON_VALVE_3_DIST_REQ )
      wire#w4
      Coil( #DATA_VALVE_3.SWITCH_ON_AUTO_REQUEST )
   END_RUNG
   RUNG wire#w1
      Contact( #SEQ_GLOBAL_AUTO_REQ )
      Contact( #CYCLE_FINISHED_1 )
      Contact( #CYCLE_FINISHED_2 )
   END_RUNG wire#w4
   RUNG wire#w1
      Contact( #SWITCH_ON_VALVE_4_DIST_REQ )
      wire#w5
      Coil( #DATA_VALVE_4.SWITCH_ON_AUTO_REQUEST )
   END_RUNG
   RUNG wire#w1
      Contact( #SEQ_GLOBAL_AUTO_REQ )
      Contact( #CYCLE_FINISHED_1 )
      Contact( #CYCLE_FINISHED_2 )
      Contact( #CYCLE_FINISHED_3 )
   END_RUNG wire#w5
   // the same network as SCL:
   #DATA_VALVE_1.SWITCH_ON_AUTO_REQUEST := "M_ONE" AND (#VALVE_1_AXIS_1_2_DIST_REQ OR #SEQ_GLOBAL_AUTO_REQ);
   #DATA_VALVE_2.SWITCH_ON_AUTO_REQUEST := "M_ONE" AND (#VALVE_2_AXIS_1_2_DIST_REQ OR (#SEQ_GLOBAL_AUTO_REQ AND #CYCLE_FINISHED_1));
   #DATA_VALVE_3.SWITCH_ON_AUTO_REQUEST := "M_ONE" AND (#SWITCH_ON_VALVE_3_DIST_REQ OR (#SEQ_GLOBAL_AUTO_REQ AND #CYCLE_FINISHED_1 AND #CYCLE_FINISHED_2));
   #DATA_VALVE_4.SWITCH_ON_AUTO_REQUEST := "M_ONE" AND (#SWITCH_ON_VALVE_4_DIST_REQ OR (#SEQ_GLOBAL_AUTO_REQ AND #CYCLE_FINISHED_1 AND #CYCLE_FINISHED_2 AND #CYCLE_FINISHED_3));
END_REGION

REGION Network 12: SWITCH ON TIME REQUEST
   RUNG wire#powerrail
      Contact( "M_ONE" )
      wire#w1
      I_Contact( #DATA_VALVE_1.SWITCH_ON )
      Contact( #O_BYTE_0.LUBRICATION_BY_TIME_VALVE_1 )
      { S7_Templates := "time_type := Time" } #DATA_VALVE_1.TIMER_1.TON(pt := #TIME_VALVE_1, et =>)
      Coil( #DATA_VALVE_1.SWITCH_ON_TIME_REQUEST )
   END_RUNG
   RUNG wire#w1
      I_Contact( #DATA_VALVE_2.SWITCH_ON )
      Contact( #O_BYTE_0.LUBRICATION_BY_TIME_VALVE_2 )
      { S7_Templates := "time_type := Time" } #DATA_VALVE_2.TIMER_1.TON(pt := #TIME_VALVE_2, et =>)
      Coil( #DATA_VALVE_2.SWITCH_ON_TIME_REQUEST )
   END_RUNG
   RUNG wire#w1
      I_Contact( #DATA_VALVE_3.SWITCH_ON )
      Contact( #O_BYTE_0.LUBRICATION_BY_TIME_VALVE_3 )
      { S7_Templates := "time_type := Time" } #DATA_VALVE_3.TIMER_1.TON(pt := #TIME_VALVE_3, et =>)
      Coil( #DATA_VALVE_3.SWITCH_ON_TIME_REQUEST )
   END_RUNG
   RUNG wire#w1
      I_Contact( #DATA_VALVE_4.SWITCH_ON )
      Contact( #O_BYTE_0.LUBRICATION_BY_TIME_VALVE_4 )
      { S7_Templates := "time_type := Time" } #DATA_VALVE_4.TIMER_1.TON(pt := #TIME_VALVE_4, et =>)
      Coil( #DATA_VALVE_4.SWITCH_ON_TIME_REQUEST )
   END_RUNG
   // the same network as SCL:
   #DATA_VALVE_1.TIMER_1.TON(IN := "M_ONE" AND NOT #DATA_VALVE_1.SWITCH_ON AND #O_BYTE_0.LUBRICATION_BY_TIME_VALVE_1,
                           PT := #TIME_VALVE_1);
   #DATA_VALVE_1.SWITCH_ON_TIME_REQUEST := #DATA_VALVE_1.TIMER_1.Q;
   #DATA_VALVE_2.TIMER_1.TON(IN := "M_ONE" AND NOT #DATA_VALVE_2.SWITCH_ON AND #O_BYTE_0.LUBRICATION_BY_TIME_VALVE_2,
                           PT := #TIME_VALVE_2);
   #DATA_VALVE_2.SWITCH_ON_TIME_REQUEST := #DATA_VALVE_2.TIMER_1.Q;
   #DATA_VALVE_3.TIMER_1.TON(IN := "M_ONE" AND NOT #DATA_VALVE_3.SWITCH_ON AND #O_BYTE_0.LUBRICATION_BY_TIME_VALVE_3,
                           PT := #TIME_VALVE_3);
   #DATA_VALVE_3.SWITCH_ON_TIME_REQUEST := #DATA_VALVE_3.TIMER_1.Q;
   #DATA_VALVE_4.TIMER_1.TON(IN := "M_ONE" AND NOT #DATA_VALVE_4.SWITCH_ON AND #O_BYTE_0.LUBRICATION_BY_TIME_VALVE_4,
                           PT := #TIME_VALVE_4);
   #DATA_VALVE_4.SWITCH_ON_TIME_REQUEST := #DATA_VALVE_4.TIMER_1.Q;
END_REGION

REGION Network 13: SWITCH ON GLOBAL REQUEST
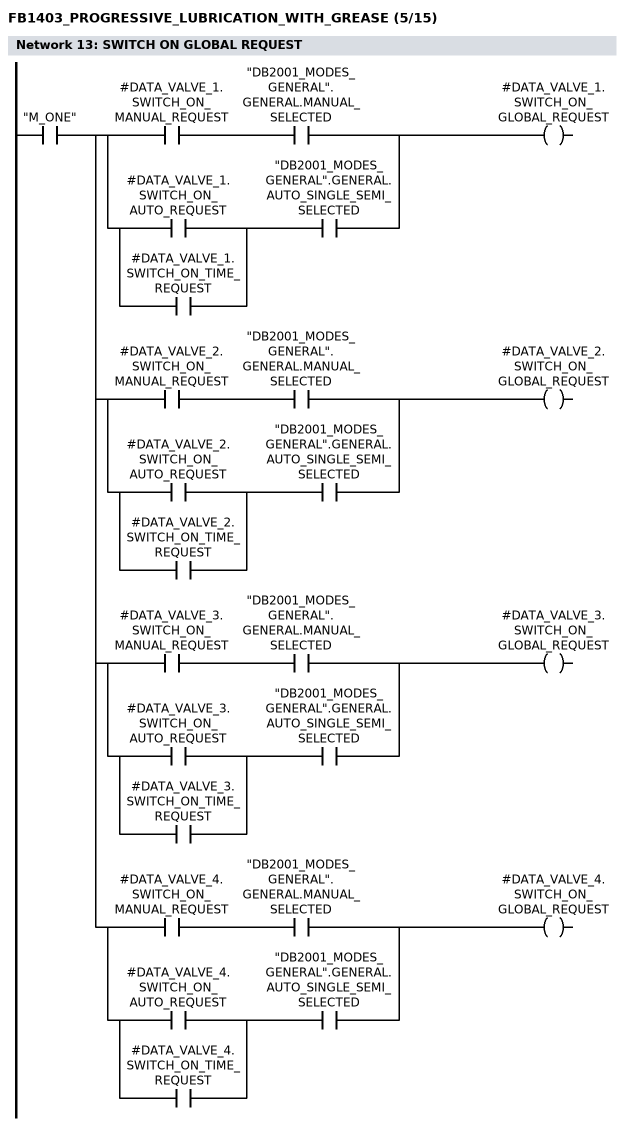
   RUNG wire#powerrail
      Contact( "M_ONE" )
      wire#w1
      Contact( #DATA_VALVE_1.SWITCH_ON_MANUAL_REQUEST )
      Contact( "DB2001_MODES_GENERAL".GENERAL.MANUAL_SELECTED )
      wire#w2
      Coil( #DATA_VALVE_1.SWITCH_ON_GLOBAL_REQUEST )
   END_RUNG
   RUNG wire#w1
      Contact( #DATA_VALVE_1.SWITCH_ON_AUTO_REQUEST )
      wire#w3
      Contact( "DB2001_MODES_GENERAL".GENERAL.AUTO_SINGLE_SEMI_SELECTED )
   END_RUNG wire#w2
   RUNG wire#w1
      Contact( #DATA_VALVE_1.SWITCH_ON_TIME_REQUEST )
   END_RUNG wire#w3
   RUNG wire#w1
      Contact( #DATA_VALVE_2.SWITCH_ON_MANUAL_REQUEST )
      Contact( "DB2001_MODES_GENERAL".GENERAL.MANUAL_SELECTED )
      wire#w4
      Coil( #DATA_VALVE_2.SWITCH_ON_GLOBAL_REQUEST )
   END_RUNG
   RUNG wire#w1
      Contact( #DATA_VALVE_2.SWITCH_ON_AUTO_REQUEST )
      wire#w5
      Contact( "DB2001_MODES_GENERAL".GENERAL.AUTO_SINGLE_SEMI_SELECTED )
   END_RUNG wire#w4
   RUNG wire#w1
      Contact( #DATA_VALVE_2.SWITCH_ON_TIME_REQUEST )
   END_RUNG wire#w5
   RUNG wire#w1
      Contact( #DATA_VALVE_3.SWITCH_ON_MANUAL_REQUEST )
      Contact( "DB2001_MODES_GENERAL".GENERAL.MANUAL_SELECTED )
      wire#w6
      Coil( #DATA_VALVE_3.SWITCH_ON_GLOBAL_REQUEST )
   END_RUNG
   RUNG wire#w1
      Contact( #DATA_VALVE_3.SWITCH_ON_AUTO_REQUEST )
      wire#w7
      Contact( "DB2001_MODES_GENERAL".GENERAL.AUTO_SINGLE_SEMI_SELECTED )
   END_RUNG wire#w6
   RUNG wire#w1
      Contact( #DATA_VALVE_3.SWITCH_ON_TIME_REQUEST )
   END_RUNG wire#w7
   RUNG wire#w1
      Contact( #DATA_VALVE_4.SWITCH_ON_MANUAL_REQUEST )
      Contact( "DB2001_MODES_GENERAL".GENERAL.MANUAL_SELECTED )
      wire#w8
      Coil( #DATA_VALVE_4.SWITCH_ON_GLOBAL_REQUEST )
   END_RUNG
   RUNG wire#w1
      Contact( #DATA_VALVE_4.SWITCH_ON_AUTO_REQUEST )
      wire#w9
      Contact( "DB2001_MODES_GENERAL".GENERAL.AUTO_SINGLE_SEMI_SELECTED )
   END_RUNG wire#w8
   RUNG wire#w1
      Contact( #DATA_VALVE_4.SWITCH_ON_TIME_REQUEST )
   END_RUNG wire#w9
   // the same network as SCL:
   #DATA_VALVE_1.SWITCH_ON_GLOBAL_REQUEST := "M_ONE" AND ((#DATA_VALVE_1.SWITCH_ON_MANUAL_REQUEST AND "DB2001_MODES_GENERAL".GENERAL.MANUAL_SELECTED) OR ((#DATA_VALVE_1.SWITCH_ON_AUTO_REQUEST OR #DATA_VALVE_1.SWITCH_ON_TIME_REQUEST) AND "DB2001_MODES_GENERAL".GENERAL.AUTO_SINGLE_SEMI_SELECTED));
   #DATA_VALVE_2.SWITCH_ON_GLOBAL_REQUEST := "M_ONE" AND ((#DATA_VALVE_2.SWITCH_ON_MANUAL_REQUEST AND "DB2001_MODES_GENERAL".GENERAL.MANUAL_SELECTED) OR ((#DATA_VALVE_2.SWITCH_ON_AUTO_REQUEST OR #DATA_VALVE_2.SWITCH_ON_TIME_REQUEST) AND "DB2001_MODES_GENERAL".GENERAL.AUTO_SINGLE_SEMI_SELECTED));
   #DATA_VALVE_3.SWITCH_ON_GLOBAL_REQUEST := "M_ONE" AND ((#DATA_VALVE_3.SWITCH_ON_MANUAL_REQUEST AND "DB2001_MODES_GENERAL".GENERAL.MANUAL_SELECTED) OR ((#DATA_VALVE_3.SWITCH_ON_AUTO_REQUEST OR #DATA_VALVE_3.SWITCH_ON_TIME_REQUEST) AND "DB2001_MODES_GENERAL".GENERAL.AUTO_SINGLE_SEMI_SELECTED));
   #DATA_VALVE_4.SWITCH_ON_GLOBAL_REQUEST := "M_ONE" AND ((#DATA_VALVE_4.SWITCH_ON_MANUAL_REQUEST AND "DB2001_MODES_GENERAL".GENERAL.MANUAL_SELECTED) OR ((#DATA_VALVE_4.SWITCH_ON_AUTO_REQUEST OR #DATA_VALVE_4.SWITCH_ON_TIME_REQUEST) AND "DB2001_MODES_GENERAL".GENERAL.AUTO_SINGLE_SEMI_SELECTED));
END_REGION

REGION Network 14: SWITCH ON COMMAND
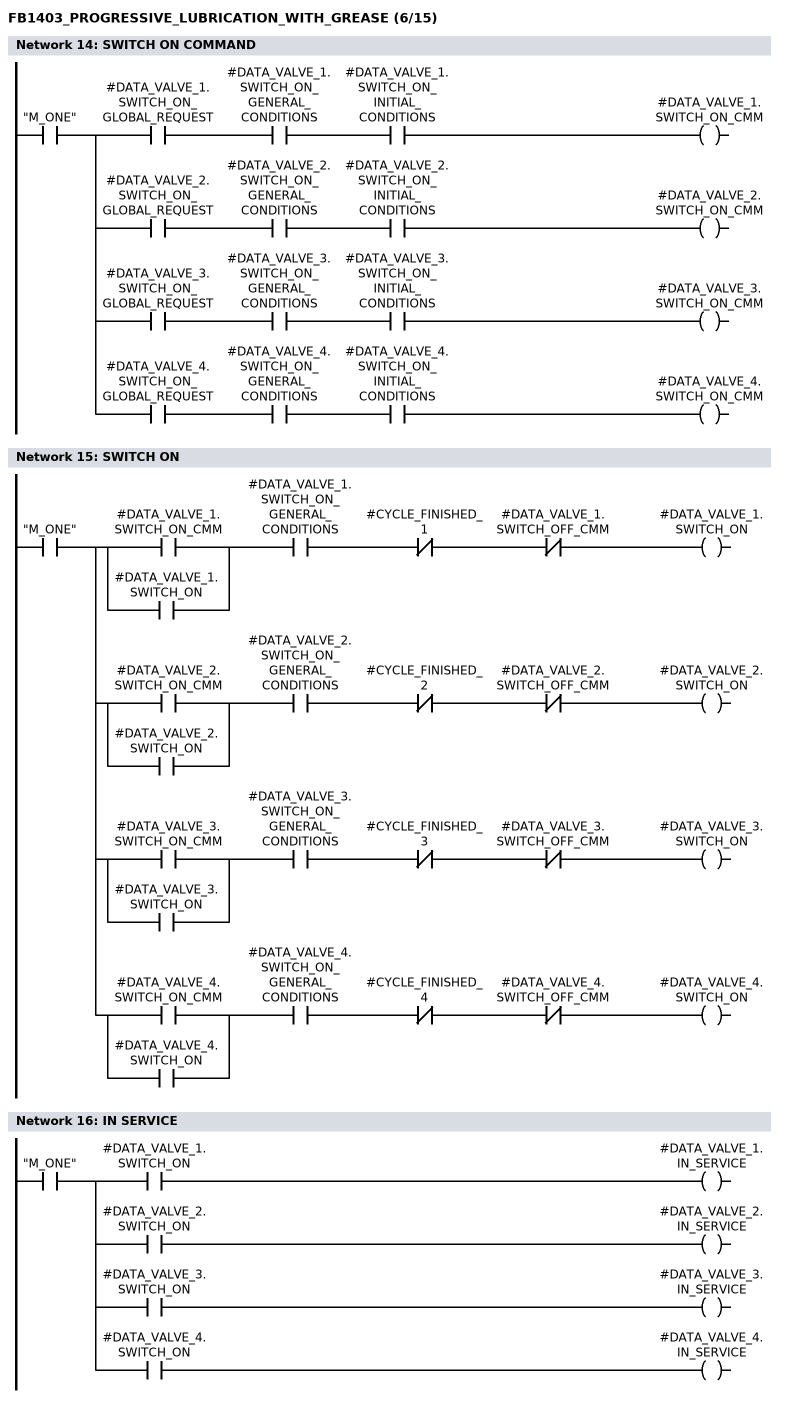
   RUNG wire#powerrail
      Contact( "M_ONE" )
      wire#w1
      Contact( #DATA_VALVE_1.SWITCH_ON_GLOBAL_REQUEST )
      Contact( #DATA_VALVE_1.SWITCH_ON_GENERAL_CONDITIONS )
      Contact( #DATA_VALVE_1.SWITCH_ON_INITIAL_CONDITIONS )
      Coil( #DATA_VALVE_1.SWITCH_ON_CMM )
   END_RUNG
   RUNG wire#w1
      Contact( #DATA_VALVE_2.SWITCH_ON_GLOBAL_REQUEST )
      Contact( #DATA_VALVE_2.SWITCH_ON_GENERAL_CONDITIONS )
      Contact( #DATA_VALVE_2.SWITCH_ON_INITIAL_CONDITIONS )
      Coil( #DATA_VALVE_2.SWITCH_ON_CMM )
   END_RUNG
   RUNG wire#w1
      Contact( #DATA_VALVE_3.SWITCH_ON_GLOBAL_REQUEST )
      Contact( #DATA_VALVE_3.SWITCH_ON_GENERAL_CONDITIONS )
      Contact( #DATA_VALVE_3.SWITCH_ON_INITIAL_CONDITIONS )
      Coil( #DATA_VALVE_3.SWITCH_ON_CMM )
   END_RUNG
   RUNG wire#w1
      Contact( #DATA_VALVE_4.SWITCH_ON_GLOBAL_REQUEST )
      Contact( #DATA_VALVE_4.SWITCH_ON_GENERAL_CONDITIONS )
      Contact( #DATA_VALVE_4.SWITCH_ON_INITIAL_CONDITIONS )
      Coil( #DATA_VALVE_4.SWITCH_ON_CMM )
   END_RUNG
   // the same network as SCL:
   #DATA_VALVE_1.SWITCH_ON_CMM := "M_ONE" AND #DATA_VALVE_1.SWITCH_ON_GLOBAL_REQUEST AND #DATA_VALVE_1.SWITCH_ON_GENERAL_CONDITIONS AND #DATA_VALVE_1.SWITCH_ON_INITIAL_CONDITIONS;
   #DATA_VALVE_2.SWITCH_ON_CMM := "M_ONE" AND #DATA_VALVE_2.SWITCH_ON_GLOBAL_REQUEST AND #DATA_VALVE_2.SWITCH_ON_GENERAL_CONDITIONS AND #DATA_VALVE_2.SWITCH_ON_INITIAL_CONDITIONS;
   #DATA_VALVE_3.SWITCH_ON_CMM := "M_ONE" AND #DATA_VALVE_3.SWITCH_ON_GLOBAL_REQUEST AND #DATA_VALVE_3.SWITCH_ON_GENERAL_CONDITIONS AND #DATA_VALVE_3.SWITCH_ON_INITIAL_CONDITIONS;
   #DATA_VALVE_4.SWITCH_ON_CMM := "M_ONE" AND #DATA_VALVE_4.SWITCH_ON_GLOBAL_REQUEST AND #DATA_VALVE_4.SWITCH_ON_GENERAL_CONDITIONS AND #DATA_VALVE_4.SWITCH_ON_INITIAL_CONDITIONS;
END_REGION

REGION Network 15: SWITCH ON
   RUNG wire#powerrail
      Contact( "M_ONE" )
      wire#w1
      Contact( #DATA_VALVE_1.SWITCH_ON_CMM )
      wire#w2
      Contact( #DATA_VALVE_1.SWITCH_ON_GENERAL_CONDITIONS )
      I_Contact( #CYCLE_FINISHED_1 )
      I_Contact( #DATA_VALVE_1.SWITCH_OFF_CMM )
      Coil( #DATA_VALVE_1.SWITCH_ON )
   END_RUNG
   RUNG wire#w1
      Contact( #DATA_VALVE_1.SWITCH_ON )
   END_RUNG wire#w2
   RUNG wire#w1
      Contact( #DATA_VALVE_2.SWITCH_ON_CMM )
      wire#w3
      Contact( #DATA_VALVE_2.SWITCH_ON_GENERAL_CONDITIONS )
      I_Contact( #CYCLE_FINISHED_2 )
      I_Contact( #DATA_VALVE_2.SWITCH_OFF_CMM )
      Coil( #DATA_VALVE_2.SWITCH_ON )
   END_RUNG
   RUNG wire#w1
      Contact( #DATA_VALVE_2.SWITCH_ON )
   END_RUNG wire#w3
   RUNG wire#w1
      Contact( #DATA_VALVE_3.SWITCH_ON_CMM )
      wire#w4
      Contact( #DATA_VALVE_3.SWITCH_ON_GENERAL_CONDITIONS )
      I_Contact( #CYCLE_FINISHED_3 )
      I_Contact( #DATA_VALVE_3.SWITCH_OFF_CMM )
      Coil( #DATA_VALVE_3.SWITCH_ON )
   END_RUNG
   RUNG wire#w1
      Contact( #DATA_VALVE_3.SWITCH_ON )
   END_RUNG wire#w4
   RUNG wire#w1
      Contact( #DATA_VALVE_4.SWITCH_ON_CMM )
      wire#w5
      Contact( #DATA_VALVE_4.SWITCH_ON_GENERAL_CONDITIONS )
      I_Contact( #CYCLE_FINISHED_4 )
      I_Contact( #DATA_VALVE_4.SWITCH_OFF_CMM )
      Coil( #DATA_VALVE_4.SWITCH_ON )
   END_RUNG
   RUNG wire#w1
      Contact( #DATA_VALVE_4.SWITCH_ON )
   END_RUNG wire#w5
   // the same network as SCL:
   #DATA_VALVE_1.SWITCH_ON := "M_ONE" AND (#DATA_VALVE_1.SWITCH_ON_CMM OR #DATA_VALVE_1.SWITCH_ON) AND #DATA_VALVE_1.SWITCH_ON_GENERAL_CONDITIONS AND NOT #CYCLE_FINISHED_1 AND NOT #DATA_VALVE_1.SWITCH_OFF_CMM;
   #DATA_VALVE_2.SWITCH_ON := "M_ONE" AND (#DATA_VALVE_2.SWITCH_ON_CMM OR #DATA_VALVE_2.SWITCH_ON) AND #DATA_VALVE_2.SWITCH_ON_GENERAL_CONDITIONS AND NOT #CYCLE_FINISHED_2 AND NOT #DATA_VALVE_2.SWITCH_OFF_CMM;
   #DATA_VALVE_3.SWITCH_ON := "M_ONE" AND (#DATA_VALVE_3.SWITCH_ON_CMM OR #DATA_VALVE_3.SWITCH_ON) AND #DATA_VALVE_3.SWITCH_ON_GENERAL_CONDITIONS AND NOT #CYCLE_FINISHED_3 AND NOT #DATA_VALVE_3.SWITCH_OFF_CMM;
   #DATA_VALVE_4.SWITCH_ON := "M_ONE" AND (#DATA_VALVE_4.SWITCH_ON_CMM OR #DATA_VALVE_4.SWITCH_ON) AND #DATA_VALVE_4.SWITCH_ON_GENERAL_CONDITIONS AND NOT #CYCLE_FINISHED_4 AND NOT #DATA_VALVE_4.SWITCH_OFF_CMM;
END_REGION

REGION Network 16: IN SERVICE
   RUNG wire#powerrail
      Contact( "M_ONE" )
      wire#w1
      Contact( #DATA_VALVE_1.SWITCH_ON )
      Coil( #DATA_VALVE_1.IN_SERVICE )
   END_RUNG
   RUNG wire#w1
      Contact( #DATA_VALVE_2.SWITCH_ON )
      Coil( #DATA_VALVE_2.IN_SERVICE )
   END_RUNG
   RUNG wire#w1
      Contact( #DATA_VALVE_3.SWITCH_ON )
      Coil( #DATA_VALVE_3.IN_SERVICE )
   END_RUNG
   RUNG wire#w1
      Contact( #DATA_VALVE_4.SWITCH_ON )
      Coil( #DATA_VALVE_4.IN_SERVICE )
   END_RUNG
   // the same network as SCL:
   #DATA_VALVE_1.IN_SERVICE := "M_ONE" AND #DATA_VALVE_1.SWITCH_ON;
   #DATA_VALVE_2.IN_SERVICE := "M_ONE" AND #DATA_VALVE_2.SWITCH_ON;
   #DATA_VALVE_3.IN_SERVICE := "M_ONE" AND #DATA_VALVE_3.SWITCH_ON;
   #DATA_VALVE_4.IN_SERVICE := "M_ONE" AND #DATA_VALVE_4.SWITCH_ON;
END_REGION

REGION Network 17: CYCLE FINISHED 1
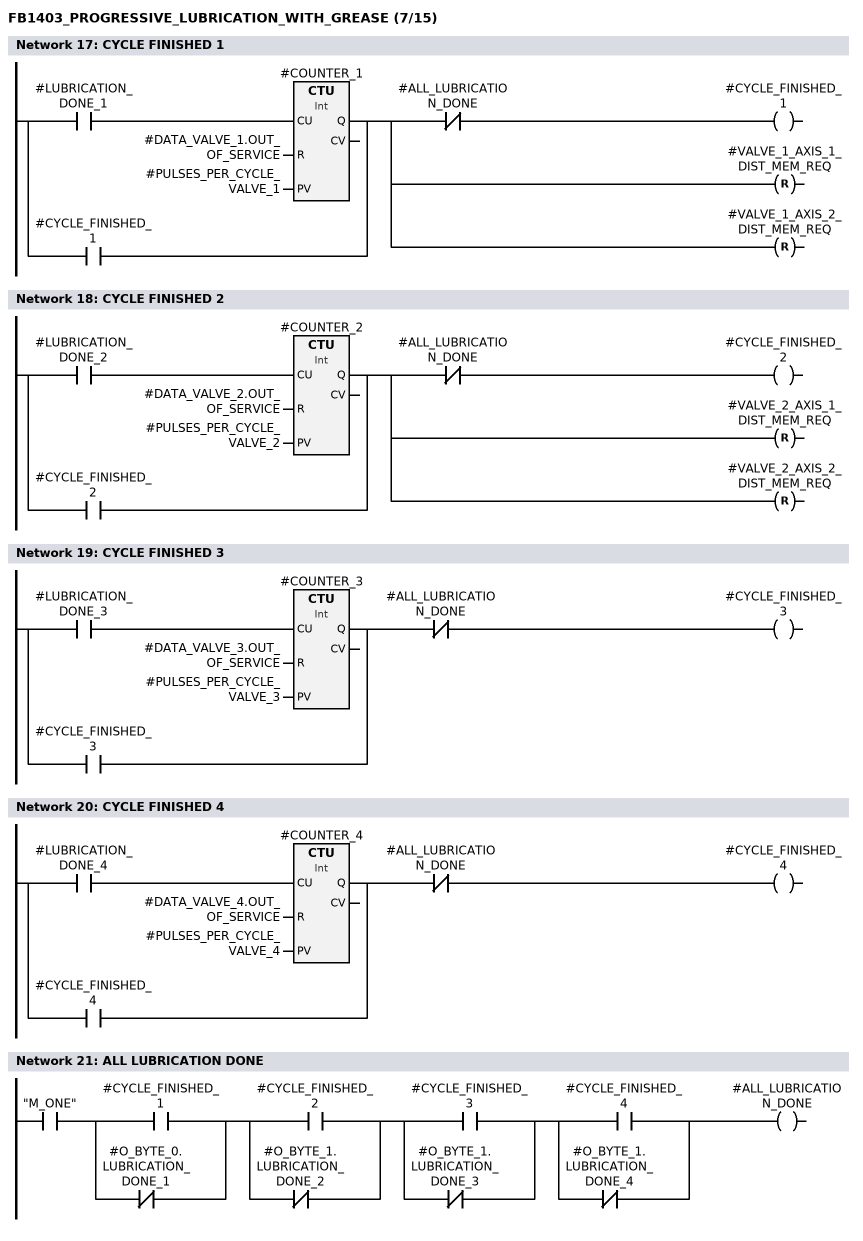
   RUNG wire#powerrail
      Contact( #LUBRICATION_DONE_1 )
      { S7_Templates := "value_type := Int" } #COUNTER_1.CTU(r := #DATA_VALVE_1.OUT_OF_SERVICE, pv := #PULSES_PER_CYCLE_VALVE_1, cv =>)
      wire#w1
      I_Contact( #ALL_LUBRICATION_DONE )
      Coil( #CYCLE_FINISHED_1 )
   END_RUNG
   RUNG wire#powerrail
      Contact( #CYCLE_FINISHED_1 )
   END_RUNG wire#w1
   RUNG wire#w1
      R_Coil( #VALVE_1_AXIS_1_DIST_MEM_REQ )
   END_RUNG
   RUNG wire#w1
      R_Coil( #VALVE_1_AXIS_2_DIST_MEM_REQ )
   END_RUNG
   // the same network as SCL:
   #COUNTER_1(CU := #LUBRICATION_DONE_1, R := #DATA_VALVE_1.OUT_OF_SERVICE, PV := #PULSES_PER_CYCLE_VALVE_1);   // CTU
   #_w1 := #COUNTER_1.Q OR #CYCLE_FINISHED_1;
   #CYCLE_FINISHED_1 := #_w1 AND NOT #ALL_LUBRICATION_DONE;
   IF #_w1 THEN
       #VALVE_1_AXIS_1_DIST_MEM_REQ := FALSE;
       #VALVE_1_AXIS_2_DIST_MEM_REQ := FALSE;
   END_IF;
END_REGION

REGION Network 18: CYCLE FINISHED 2
   RUNG wire#powerrail
      Contact( #LUBRICATION_DONE_2 )
      { S7_Templates := "value_type := Int" } #COUNTER_2.CTU(r := #DATA_VALVE_2.OUT_OF_SERVICE, pv := #PULSES_PER_CYCLE_VALVE_2, cv =>)
      wire#w1
      I_Contact( #ALL_LUBRICATION_DONE )
      Coil( #CYCLE_FINISHED_2 )
   END_RUNG
   RUNG wire#powerrail
      Contact( #CYCLE_FINISHED_2 )
   END_RUNG wire#w1
   RUNG wire#w1
      R_Coil( #VALVE_2_AXIS_1_DIST_MEM_REQ )
   END_RUNG
   RUNG wire#w1
      R_Coil( #VALVE_2_AXIS_2_DIST_MEM_REQ )
   END_RUNG
   // the same network as SCL:
   #COUNTER_2(CU := #LUBRICATION_DONE_2, R := #DATA_VALVE_2.OUT_OF_SERVICE, PV := #PULSES_PER_CYCLE_VALVE_2);   // CTU
   #_w1 := #COUNTER_2.Q OR #CYCLE_FINISHED_2;
   #CYCLE_FINISHED_2 := #_w1 AND NOT #ALL_LUBRICATION_DONE;
   IF #_w1 THEN
       #VALVE_2_AXIS_1_DIST_MEM_REQ := FALSE;
       #VALVE_2_AXIS_2_DIST_MEM_REQ := FALSE;
   END_IF;
END_REGION

REGION Network 19: CYCLE FINISHED 3
   RUNG wire#powerrail
      Contact( #LUBRICATION_DONE_3 )
      { S7_Templates := "value_type := Int" } #COUNTER_3.CTU(r := #DATA_VALVE_3.OUT_OF_SERVICE, pv := #PULSES_PER_CYCLE_VALVE_3, cv =>)
      wire#w1
      I_Contact( #ALL_LUBRICATION_DONE )
      Coil( #CYCLE_FINISHED_3 )
   END_RUNG
   RUNG wire#powerrail
      Contact( #CYCLE_FINISHED_3 )
   END_RUNG wire#w1
   // the same network as SCL:
   #COUNTER_3(CU := #LUBRICATION_DONE_3, R := #DATA_VALVE_3.OUT_OF_SERVICE, PV := #PULSES_PER_CYCLE_VALVE_3);   // CTU
   #CYCLE_FINISHED_3 := (#COUNTER_3.Q OR #CYCLE_FINISHED_3) AND NOT #ALL_LUBRICATION_DONE;
END_REGION

REGION Network 20: CYCLE FINISHED 4
   RUNG wire#powerrail
      Contact( #LUBRICATION_DONE_4 )
      { S7_Templates := "value_type := Int" } #COUNTER_4.CTU(r := #DATA_VALVE_4.OUT_OF_SERVICE, pv := #PULSES_PER_CYCLE_VALVE_4, cv =>)
      wire#w1
      I_Contact( #ALL_LUBRICATION_DONE )
      Coil( #CYCLE_FINISHED_4 )
   END_RUNG
   RUNG wire#powerrail
      Contact( #CYCLE_FINISHED_4 )
   END_RUNG wire#w1
   // the same network as SCL:
   #COUNTER_4(CU := #LUBRICATION_DONE_4, R := #DATA_VALVE_4.OUT_OF_SERVICE, PV := #PULSES_PER_CYCLE_VALVE_4);   // CTU
   #CYCLE_FINISHED_4 := (#COUNTER_4.Q OR #CYCLE_FINISHED_4) AND NOT #ALL_LUBRICATION_DONE;
END_REGION

REGION Network 21: ALL LUBRICATION DONE
   RUNG wire#powerrail
      Contact( "M_ONE" )
      wire#w1
      Contact( #CYCLE_FINISHED_1 )
      wire#w2
      Contact( #CYCLE_FINISHED_2 )
      wire#w3
      Contact( #CYCLE_FINISHED_3 )
      wire#w4
      Contact( #CYCLE_FINISHED_4 )
      wire#w5
      Coil( #ALL_LUBRICATION_DONE )
   END_RUNG
   RUNG wire#w1
      I_Contact( #O_BYTE_0.LUBRICATION_DONE_1 )
   END_RUNG wire#w2
   RUNG wire#w2
      I_Contact( #O_BYTE_1.LUBRICATION_DONE_2 )
   END_RUNG wire#w3
   RUNG wire#w3
      I_Contact( #O_BYTE_1.LUBRICATION_DONE_3 )
   END_RUNG wire#w4
   RUNG wire#w4
      I_Contact( #O_BYTE_1.LUBRICATION_DONE_4 )
   END_RUNG wire#w5
   // the same network as SCL:
   #ALL_LUBRICATION_DONE := "M_ONE" AND (#CYCLE_FINISHED_1 OR NOT #O_BYTE_0.LUBRICATION_DONE_1) AND (#CYCLE_FINISHED_2 OR NOT #O_BYTE_1.LUBRICATION_DONE_2) AND (#CYCLE_FINISHED_3 OR NOT #O_BYTE_1.LUBRICATION_DONE_3) AND (#CYCLE_FINISHED_4 OR NOT #O_BYTE_1.LUBRICATION_DONE_4);
END_REGION

REGION Network 22: SWITCH OFF GENERAL CONDITIONS
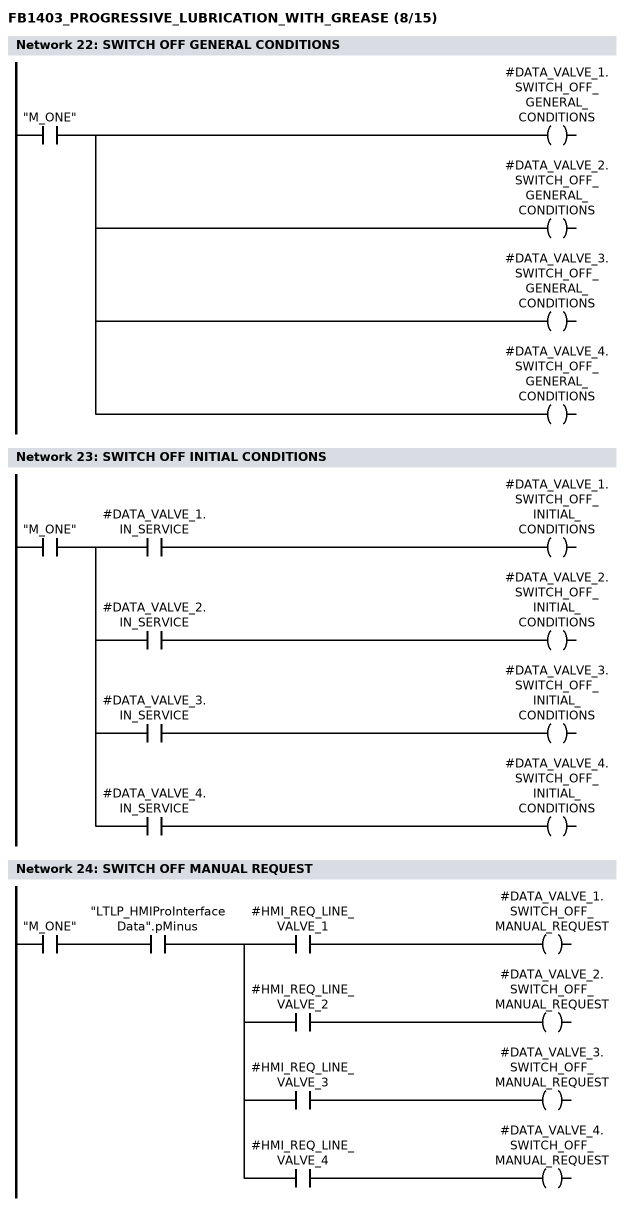
   RUNG wire#powerrail
      Contact( "M_ONE" )
      wire#w1
      Coil( #DATA_VALVE_1.SWITCH_OFF_GENERAL_CONDITIONS )
   END_RUNG
   RUNG wire#w1
      Coil( #DATA_VALVE_2.SWITCH_OFF_GENERAL_CONDITIONS )
   END_RUNG
   RUNG wire#w1
      Coil( #DATA_VALVE_3.SWITCH_OFF_GENERAL_CONDITIONS )
   END_RUNG
   RUNG wire#w1
      Coil( #DATA_VALVE_4.SWITCH_OFF_GENERAL_CONDITIONS )
   END_RUNG
   // the same network as SCL:
   #DATA_VALVE_1.SWITCH_OFF_GENERAL_CONDITIONS := "M_ONE";
   #DATA_VALVE_2.SWITCH_OFF_GENERAL_CONDITIONS := "M_ONE";
   #DATA_VALVE_3.SWITCH_OFF_GENERAL_CONDITIONS := "M_ONE";
   #DATA_VALVE_4.SWITCH_OFF_GENERAL_CONDITIONS := "M_ONE";
END_REGION

REGION Network 23: SWITCH OFF INITIAL CONDITIONS
   RUNG wire#powerrail
      Contact( "M_ONE" )
      wire#w1
      Contact( #DATA_VALVE_1.IN_SERVICE )
      Coil( #DATA_VALVE_1.SWITCH_OFF_INITIAL_CONDITIONS )
   END_RUNG
   RUNG wire#w1
      Contact( #DATA_VALVE_2.IN_SERVICE )
      Coil( #DATA_VALVE_2.SWITCH_OFF_INITIAL_CONDITIONS )
   END_RUNG
   RUNG wire#w1
      Contact( #DATA_VALVE_3.IN_SERVICE )
      Coil( #DATA_VALVE_3.SWITCH_OFF_INITIAL_CONDITIONS )
   END_RUNG
   RUNG wire#w1
      Contact( #DATA_VALVE_4.IN_SERVICE )
      Coil( #DATA_VALVE_4.SWITCH_OFF_INITIAL_CONDITIONS )
   END_RUNG
   // the same network as SCL:
   #DATA_VALVE_1.SWITCH_OFF_INITIAL_CONDITIONS := "M_ONE" AND #DATA_VALVE_1.IN_SERVICE;
   #DATA_VALVE_2.SWITCH_OFF_INITIAL_CONDITIONS := "M_ONE" AND #DATA_VALVE_2.IN_SERVICE;
   #DATA_VALVE_3.SWITCH_OFF_INITIAL_CONDITIONS := "M_ONE" AND #DATA_VALVE_3.IN_SERVICE;
   #DATA_VALVE_4.SWITCH_OFF_INITIAL_CONDITIONS := "M_ONE" AND #DATA_VALVE_4.IN_SERVICE;
END_REGION

REGION Network 24: SWITCH OFF MANUAL REQUEST
   RUNG wire#powerrail
      Contact( "M_ONE" )
      Contact( "LTLP_HMIProInterfaceData".pMinus )
      wire#w1
      Contact( #HMI_REQ_LINE_VALVE_1 )
      Coil( #DATA_VALVE_1.SWITCH_OFF_MANUAL_REQUEST )
   END_RUNG
   RUNG wire#w1
      Contact( #HMI_REQ_LINE_VALVE_2 )
      Coil( #DATA_VALVE_2.SWITCH_OFF_MANUAL_REQUEST )
   END_RUNG
   RUNG wire#w1
      Contact( #HMI_REQ_LINE_VALVE_3 )
      Coil( #DATA_VALVE_3.SWITCH_OFF_MANUAL_REQUEST )
   END_RUNG
   RUNG wire#w1
      Contact( #HMI_REQ_LINE_VALVE_4 )
      Coil( #DATA_VALVE_4.SWITCH_OFF_MANUAL_REQUEST )
   END_RUNG
   // the same network as SCL:
   #_w1 := "M_ONE" AND "LTLP_HMIProInterfaceData".pMinus;
   #DATA_VALVE_1.SWITCH_OFF_MANUAL_REQUEST := #_w1 AND #HMI_REQ_LINE_VALVE_1;
   #DATA_VALVE_2.SWITCH_OFF_MANUAL_REQUEST := #_w1 AND #HMI_REQ_LINE_VALVE_2;
   #DATA_VALVE_3.SWITCH_OFF_MANUAL_REQUEST := #_w1 AND #HMI_REQ_LINE_VALVE_3;
   #DATA_VALVE_4.SWITCH_OFF_MANUAL_REQUEST := #_w1 AND #HMI_REQ_LINE_VALVE_4;
END_REGION

REGION Network 25: SWITCH OFF AUTO REQUEST
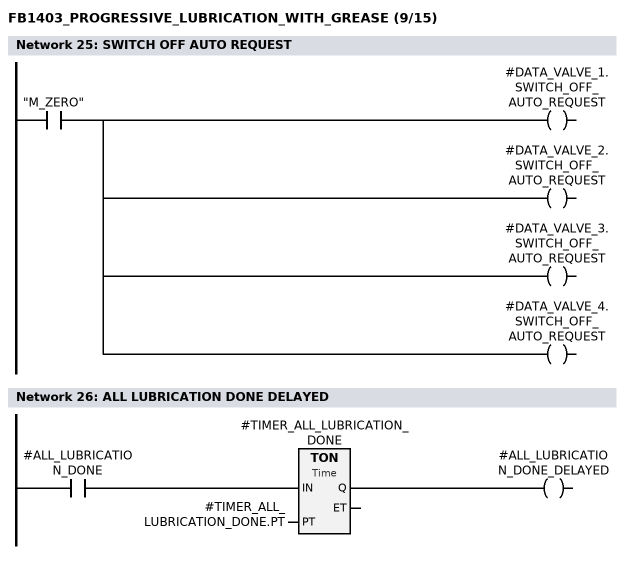
   RUNG wire#powerrail
      Contact( "M_ZERO" )
      wire#w1
      Coil( #DATA_VALVE_1.SWITCH_OFF_AUTO_REQUEST )
   END_RUNG
   RUNG wire#w1
      Coil( #DATA_VALVE_2.SWITCH_OFF_AUTO_REQUEST )
   END_RUNG
   RUNG wire#w1
      Coil( #DATA_VALVE_3.SWITCH_OFF_AUTO_REQUEST )
   END_RUNG
   RUNG wire#w1
      Coil( #DATA_VALVE_4.SWITCH_OFF_AUTO_REQUEST )
   END_RUNG
   // the same network as SCL:
   #DATA_VALVE_1.SWITCH_OFF_AUTO_REQUEST := "M_ZERO";
   #DATA_VALVE_2.SWITCH_OFF_AUTO_REQUEST := "M_ZERO";
   #DATA_VALVE_3.SWITCH_OFF_AUTO_REQUEST := "M_ZERO";
   #DATA_VALVE_4.SWITCH_OFF_AUTO_REQUEST := "M_ZERO";
END_REGION

REGION Network 26: ALL LUBRICATION DONE DELAYED
   RUNG wire#powerrail
      Contact( #ALL_LUBRICATION_DONE )
      { S7_Templates := "time_type := Time" } #TIMER_ALL_LUBRICATION_DONE.TON(pt := #TIMER_ALL_LUBRICATION_DONE.PT, et =>)
      Coil( #ALL_LUBRICATION_DONE_DELAYED )
   END_RUNG
   // the same network as SCL:
   #TIMER_ALL_LUBRICATION_DONE(IN := #ALL_LUBRICATION_DONE, PT := #TIMER_ALL_LUBRICATION_DONE.PT);   // TON
   #ALL_LUBRICATION_DONE_DELAYED := #TIMER_ALL_LUBRICATION_DONE.Q;
END_REGION

REGION Network 27: SWITCH OFF GLOBAL REQUEST
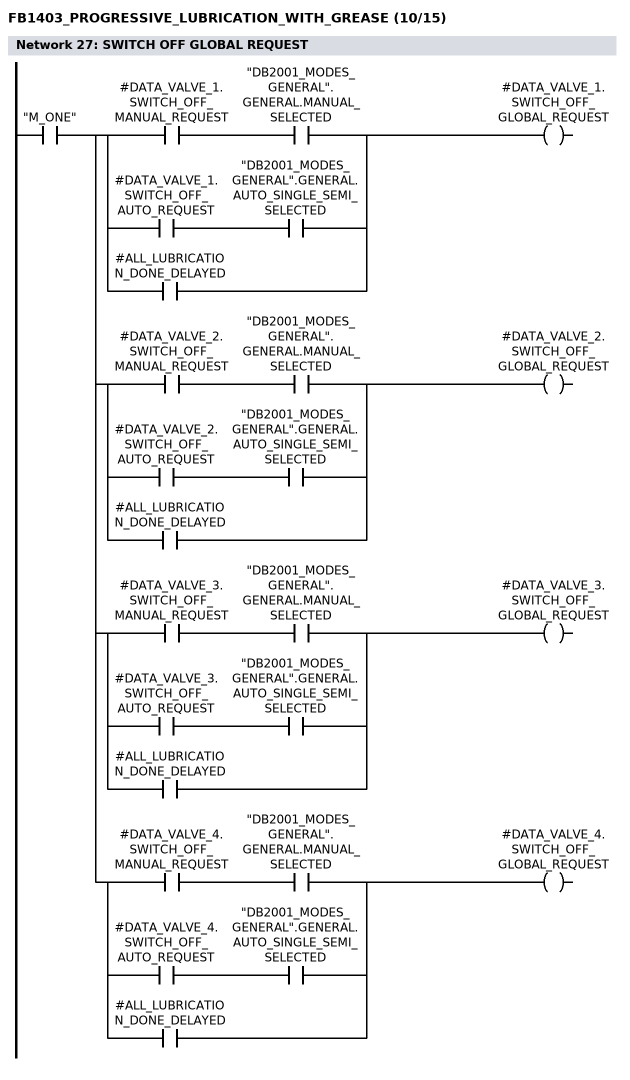
   RUNG wire#powerrail
      Contact( "M_ONE" )
      wire#w1
      Contact( #DATA_VALVE_1.SWITCH_OFF_MANUAL_REQUEST )
      Contact( "DB2001_MODES_GENERAL".GENERAL.MANUAL_SELECTED )
      wire#w2
      Coil( #DATA_VALVE_1.SWITCH_OFF_GLOBAL_REQUEST )
   END_RUNG
   RUNG wire#w1
      Contact( #DATA_VALVE_1.SWITCH_OFF_AUTO_REQUEST )
      Contact( "DB2001_MODES_GENERAL".GENERAL.AUTO_SINGLE_SEMI_SELECTED )
   END_RUNG wire#w2
   RUNG wire#w1
      Contact( #ALL_LUBRICATION_DONE_DELAYED )
   END_RUNG wire#w2
   RUNG wire#w1
      Contact( #DATA_VALVE_2.SWITCH_OFF_MANUAL_REQUEST )
      Contact( "DB2001_MODES_GENERAL".GENERAL.MANUAL_SELECTED )
      wire#w3
      Coil( #DATA_VALVE_2.SWITCH_OFF_GLOBAL_REQUEST )
   END_RUNG
   RUNG wire#w1
      Contact( #DATA_VALVE_2.SWITCH_OFF_AUTO_REQUEST )
      Contact( "DB2001_MODES_GENERAL".GENERAL.AUTO_SINGLE_SEMI_SELECTED )
   END_RUNG wire#w3
   RUNG wire#w1
      Contact( #ALL_LUBRICATION_DONE_DELAYED )
   END_RUNG wire#w3
   RUNG wire#w1
      Contact( #DATA_VALVE_3.SWITCH_OFF_MANUAL_REQUEST )
      Contact( "DB2001_MODES_GENERAL".GENERAL.MANUAL_SELECTED )
      wire#w4
      Coil( #DATA_VALVE_3.SWITCH_OFF_GLOBAL_REQUEST )
   END_RUNG
   RUNG wire#w1
      Contact( #DATA_VALVE_3.SWITCH_OFF_AUTO_REQUEST )
      Contact( "DB2001_MODES_GENERAL".GENERAL.AUTO_SINGLE_SEMI_SELECTED )
   END_RUNG wire#w4
   RUNG wire#w1
      Contact( #ALL_LUBRICATION_DONE_DELAYED )
   END_RUNG wire#w4
   RUNG wire#w1
      Contact( #DATA_VALVE_4.SWITCH_OFF_MANUAL_REQUEST )
      Contact( "DB2001_MODES_GENERAL".GENERAL.MANUAL_SELECTED )
      wire#w5
      Coil( #DATA_VALVE_4.SWITCH_OFF_GLOBAL_REQUEST )
   END_RUNG
   RUNG wire#w1
      Contact( #DATA_VALVE_4.SWITCH_OFF_AUTO_REQUEST )
      Contact( "DB2001_MODES_GENERAL".GENERAL.AUTO_SINGLE_SEMI_SELECTED )
   END_RUNG wire#w5
   RUNG wire#w1
      Contact( #ALL_LUBRICATION_DONE_DELAYED )
   END_RUNG wire#w5
   // the same network as SCL:
   #DATA_VALVE_1.SWITCH_OFF_GLOBAL_REQUEST := "M_ONE" AND ((#DATA_VALVE_1.SWITCH_OFF_MANUAL_REQUEST AND "DB2001_MODES_GENERAL".GENERAL.MANUAL_SELECTED) OR (#DATA_VALVE_1.SWITCH_OFF_AUTO_REQUEST AND "DB2001_MODES_GENERAL".GENERAL.AUTO_SINGLE_SEMI_SELECTED) OR #ALL_LUBRICATION_DONE_DELAYED);
   #DATA_VALVE_2.SWITCH_OFF_GLOBAL_REQUEST := "M_ONE" AND ((#DATA_VALVE_2.SWITCH_OFF_MANUAL_REQUEST AND "DB2001_MODES_GENERAL".GENERAL.MANUAL_SELECTED) OR (#DATA_VALVE_2.SWITCH_OFF_AUTO_REQUEST AND "DB2001_MODES_GENERAL".GENERAL.AUTO_SINGLE_SEMI_SELECTED) OR #ALL_LUBRICATION_DONE_DELAYED);
   #DATA_VALVE_3.SWITCH_OFF_GLOBAL_REQUEST := "M_ONE" AND ((#DATA_VALVE_3.SWITCH_OFF_MANUAL_REQUEST AND "DB2001_MODES_GENERAL".GENERAL.MANUAL_SELECTED) OR (#DATA_VALVE_3.SWITCH_OFF_AUTO_REQUEST AND "DB2001_MODES_GENERAL".GENERAL.AUTO_SINGLE_SEMI_SELECTED) OR #ALL_LUBRICATION_DONE_DELAYED);
   #DATA_VALVE_4.SWITCH_OFF_GLOBAL_REQUEST := "M_ONE" AND ((#DATA_VALVE_4.SWITCH_OFF_MANUAL_REQUEST AND "DB2001_MODES_GENERAL".GENERAL.MANUAL_SELECTED) OR (#DATA_VALVE_4.SWITCH_OFF_AUTO_REQUEST AND "DB2001_MODES_GENERAL".GENERAL.AUTO_SINGLE_SEMI_SELECTED) OR #ALL_LUBRICATION_DONE_DELAYED);
END_REGION

REGION Network 28: SWITCH OFF COMMAND
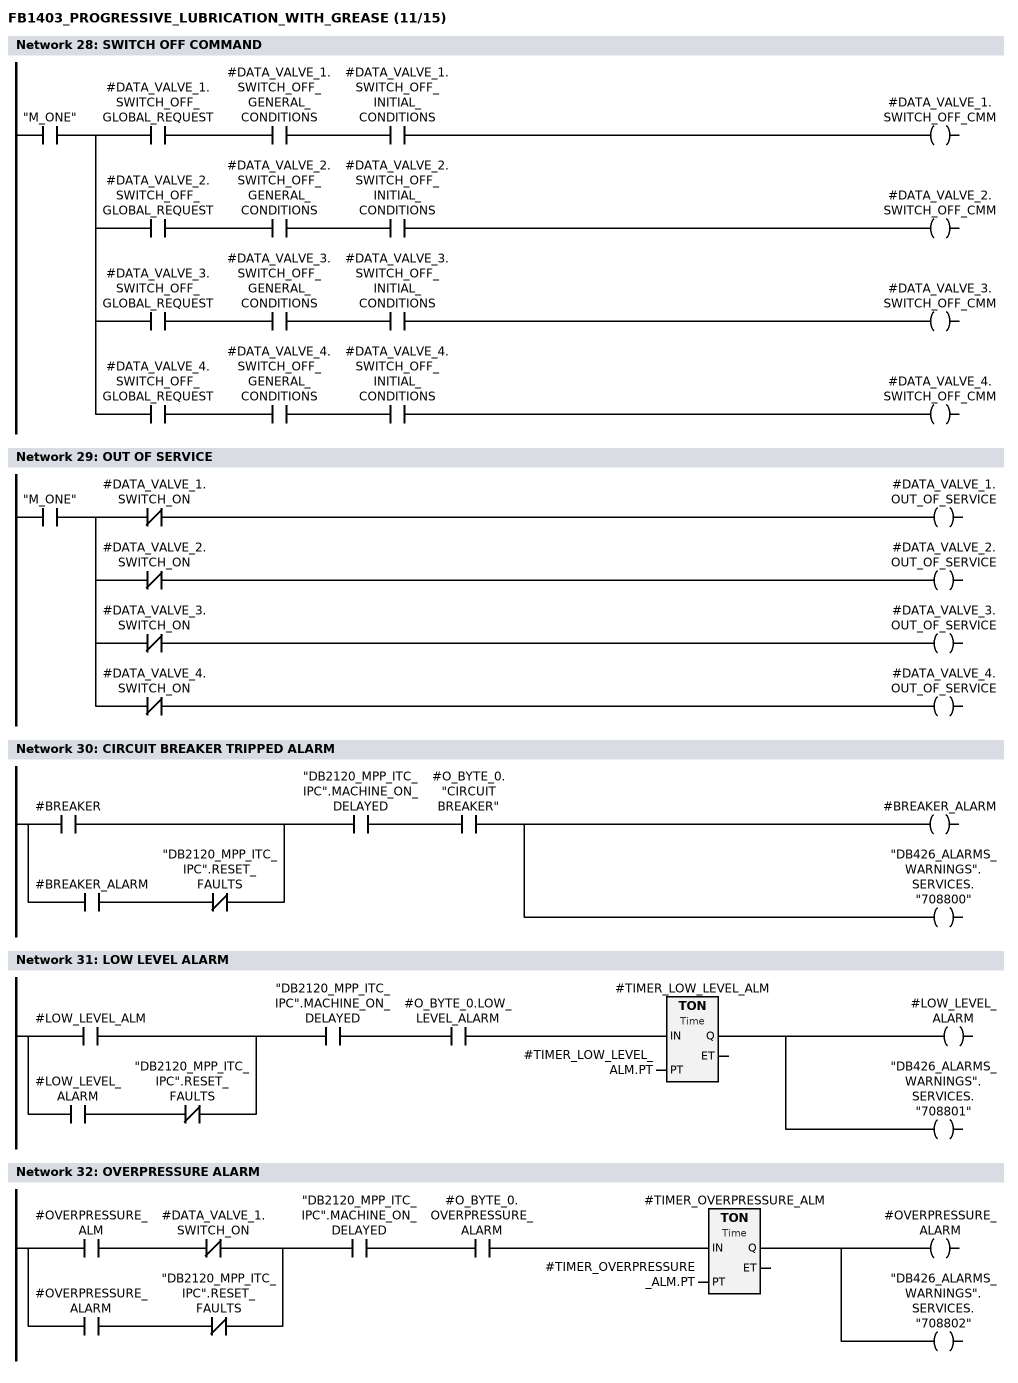
   RUNG wire#powerrail
      Contact( "M_ONE" )
      wire#w1
      Contact( #DATA_VALVE_1.SWITCH_OFF_GLOBAL_REQUEST )
      Contact( #DATA_VALVE_1.SWITCH_OFF_GENERAL_CONDITIONS )
      Contact( #DATA_VALVE_1.SWITCH_OFF_INITIAL_CONDITIONS )
      Coil( #DATA_VALVE_1.SWITCH_OFF_CMM )
   END_RUNG
   RUNG wire#w1
      Contact( #DATA_VALVE_2.SWITCH_OFF_GLOBAL_REQUEST )
      Contact( #DATA_VALVE_2.SWITCH_OFF_GENERAL_CONDITIONS )
      Contact( #DATA_VALVE_2.SWITCH_OFF_INITIAL_CONDITIONS )
      Coil( #DATA_VALVE_2.SWITCH_OFF_CMM )
   END_RUNG
   RUNG wire#w1
      Contact( #DATA_VALVE_3.SWITCH_OFF_GLOBAL_REQUEST )
      Contact( #DATA_VALVE_3.SWITCH_OFF_GENERAL_CONDITIONS )
      Contact( #DATA_VALVE_3.SWITCH_OFF_INITIAL_CONDITIONS )
      Coil( #DATA_VALVE_3.SWITCH_OFF_CMM )
   END_RUNG
   RUNG wire#w1
      Contact( #DATA_VALVE_4.SWITCH_OFF_GLOBAL_REQUEST )
      Contact( #DATA_VALVE_4.SWITCH_OFF_GENERAL_CONDITIONS )
      Contact( #DATA_VALVE_4.SWITCH_OFF_INITIAL_CONDITIONS )
      Coil( #DATA_VALVE_4.SWITCH_OFF_CMM )
   END_RUNG
   // the same network as SCL:
   #DATA_VALVE_1.SWITCH_OFF_CMM := "M_ONE" AND #DATA_VALVE_1.SWITCH_OFF_GLOBAL_REQUEST AND #DATA_VALVE_1.SWITCH_OFF_GENERAL_CONDITIONS AND #DATA_VALVE_1.SWITCH_OFF_INITIAL_CONDITIONS;
   #DATA_VALVE_2.SWITCH_OFF_CMM := "M_ONE" AND #DATA_VALVE_2.SWITCH_OFF_GLOBAL_REQUEST AND #DATA_VALVE_2.SWITCH_OFF_GENERAL_CONDITIONS AND #DATA_VALVE_2.SWITCH_OFF_INITIAL_CONDITIONS;
   #DATA_VALVE_3.SWITCH_OFF_CMM := "M_ONE" AND #DATA_VALVE_3.SWITCH_OFF_GLOBAL_REQUEST AND #DATA_VALVE_3.SWITCH_OFF_GENERAL_CONDITIONS AND #DATA_VALVE_3.SWITCH_OFF_INITIAL_CONDITIONS;
   #DATA_VALVE_4.SWITCH_OFF_CMM := "M_ONE" AND #DATA_VALVE_4.SWITCH_OFF_GLOBAL_REQUEST AND #DATA_VALVE_4.SWITCH_OFF_GENERAL_CONDITIONS AND #DATA_VALVE_4.SWITCH_OFF_INITIAL_CONDITIONS;
END_REGION

REGION Network 29: OUT OF SERVICE
   RUNG wire#powerrail
      Contact( "M_ONE" )
      wire#w1
      I_Contact( #DATA_VALVE_1.SWITCH_ON )
      Coil( #DATA_VALVE_1.OUT_OF_SERVICE )
   END_RUNG
   RUNG wire#w1
      I_Contact( #DATA_VALVE_2.SWITCH_ON )
      Coil( #DATA_VALVE_2.OUT_OF_SERVICE )
   END_RUNG
   RUNG wire#w1
      I_Contact( #DATA_VALVE_3.SWITCH_ON )
      Coil( #DATA_VALVE_3.OUT_OF_SERVICE )
   END_RUNG
   RUNG wire#w1
      I_Contact( #DATA_VALVE_4.SWITCH_ON )
      Coil( #DATA_VALVE_4.OUT_OF_SERVICE )
   END_RUNG
   // the same network as SCL:
   #DATA_VALVE_1.OUT_OF_SERVICE := "M_ONE" AND NOT #DATA_VALVE_1.SWITCH_ON;
   #DATA_VALVE_2.OUT_OF_SERVICE := "M_ONE" AND NOT #DATA_VALVE_2.SWITCH_ON;
   #DATA_VALVE_3.OUT_OF_SERVICE := "M_ONE" AND NOT #DATA_VALVE_3.SWITCH_ON;
   #DATA_VALVE_4.OUT_OF_SERVICE := "M_ONE" AND NOT #DATA_VALVE_4.SWITCH_ON;
END_REGION

REGION Network 30: CIRCUIT BREAKER TRIPPED ALARM
   RUNG wire#powerrail
      Contact( #BREAKER )
      wire#w1
      Contact( "DB2120_MPP_ITC_IPC".MACHINE_ON_DELAYED )
      Contact( #O_BYTE_0."CIRCUIT BREAKER" )
      wire#w2
      Coil( #BREAKER_ALARM )
   END_RUNG
   RUNG wire#powerrail
      Contact( #BREAKER_ALARM )
      I_Contact( "DB2120_MPP_ITC_IPC".RESET_FAULTS )
   END_RUNG wire#w1
   RUNG wire#w2
      Coil( "DB426_ALARMS_WARNINGS".SERVICES."708800" )
   END_RUNG
   // the same network as SCL:
   #BREAKER_ALARM := (#BREAKER OR (#BREAKER_ALARM AND NOT "DB2120_MPP_ITC_IPC".RESET_FAULTS)) AND "DB2120_MPP_ITC_IPC".MACHINE_ON_DELAYED AND #O_BYTE_0."CIRCUIT BREAKER";
   "DB426_ALARMS_WARNINGS".SERVICES."708800" := #BREAKER_ALARM;
END_REGION

REGION Network 31: LOW LEVEL ALARM
   RUNG wire#powerrail
      Contact( #LOW_LEVEL_ALM )
      wire#w1
      Contact( "DB2120_MPP_ITC_IPC".MACHINE_ON_DELAYED )
      Contact( #O_BYTE_0.LOW_LEVEL_ALARM )
      { S7_Templates := "time_type := Time" } #TIMER_LOW_LEVEL_ALM.TON(pt := #TIMER_LOW_LEVEL_ALM.PT, et =>)
      wire#w2
      Coil( #LOW_LEVEL_ALARM )
   END_RUNG
   RUNG wire#powerrail
      Contact( #LOW_LEVEL_ALARM )
      I_Contact( "DB2120_MPP_ITC_IPC".RESET_FAULTS )
   END_RUNG wire#w1
   RUNG wire#w2
      Coil( "DB426_ALARMS_WARNINGS".SERVICES."708801" )
   END_RUNG
   // the same network as SCL:
   #TIMER_LOW_LEVEL_ALM(IN := (#LOW_LEVEL_ALM OR (#LOW_LEVEL_ALARM AND NOT "DB2120_MPP_ITC_IPC".RESET_FAULTS)) AND "DB2120_MPP_ITC_IPC".MACHINE_ON_DELAYED AND #O_BYTE_0.LOW_LEVEL_ALARM,   // TON
                        PT := #TIMER_LOW_LEVEL_ALM.PT);
   #LOW_LEVEL_ALARM := #TIMER_LOW_LEVEL_ALM.Q;
   "DB426_ALARMS_WARNINGS".SERVICES."708801" := #TIMER_LOW_LEVEL_ALM.Q;
END_REGION

REGION Network 32: OVERPRESSURE ALARM
   RUNG wire#powerrail
      Contact( #OVERPRESSURE_ALM )
      I_Contact( #DATA_VALVE_1.SWITCH_ON )
      wire#w1
      Contact( "DB2120_MPP_ITC_IPC".MACHINE_ON_DELAYED )
      Contact( #O_BYTE_0.OVERPRESSURE_ALARM )
      { S7_Templates := "time_type := Time" } #TIMER_OVERPRESSURE_ALM.TON(pt := #TIMER_OVERPRESSURE_ALM.PT, et =>)
      wire#w2
      Coil( #OVERPRESSURE_ALARM )
   END_RUNG
   RUNG wire#powerrail
      Contact( #OVERPRESSURE_ALARM )
      I_Contact( "DB2120_MPP_ITC_IPC".RESET_FAULTS )
   END_RUNG wire#w1
   RUNG wire#w2
      Coil( "DB426_ALARMS_WARNINGS".SERVICES."708802" )
   END_RUNG
   // the same network as SCL:
   #TIMER_OVERPRESSURE_ALM(IN := ((#OVERPRESSURE_ALM AND NOT #DATA_VALVE_1.SWITCH_ON) OR (#OVERPRESSURE_ALARM AND NOT "DB2120_MPP_ITC_IPC".RESET_FAULTS)) AND "DB2120_MPP_ITC_IPC".MACHINE_ON_DELAYED AND #O_BYTE_0.OVERPRESSURE_ALARM,   // TON
                           PT := #TIMER_OVERPRESSURE_ALM.PT);
   #OVERPRESSURE_ALARM := #TIMER_OVERPRESSURE_ALM.Q;
   "DB426_ALARMS_WARNINGS".SERVICES."708802" := #TIMER_OVERPRESSURE_ALM.Q;
END_REGION

REGION Network 33: ANY CYCLE NOT DONE
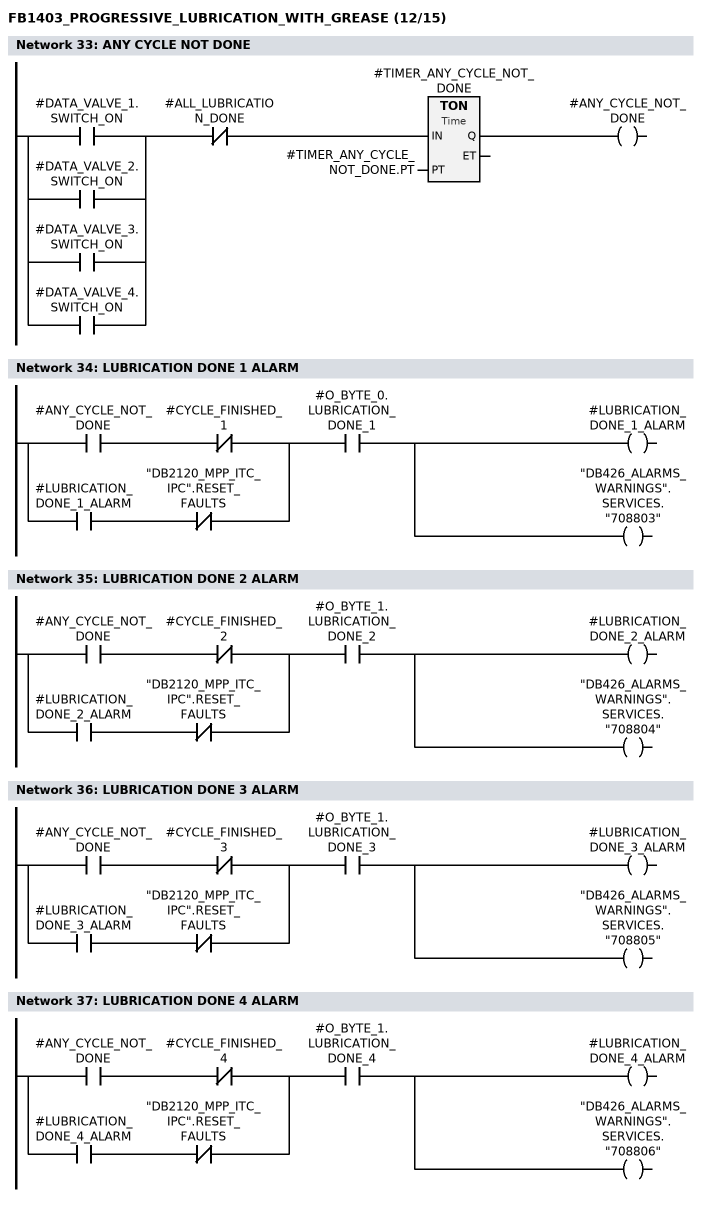
   RUNG wire#powerrail
      Contact( #DATA_VALVE_1.SWITCH_ON )
      wire#w1
      I_Contact( #ALL_LUBRICATION_DONE )
      { S7_Templates := "time_type := Time" } #TIMER_ANY_CYCLE_NOT_DONE.TON(pt := #TIMER_ANY_CYCLE_NOT_DONE.PT, et =>)
      Coil( #ANY_CYCLE_NOT_DONE )
   END_RUNG
   RUNG wire#powerrail
      Contact( #DATA_VALVE_2.SWITCH_ON )
   END_RUNG wire#w1
   RUNG wire#powerrail
      Contact( #DATA_VALVE_3.SWITCH_ON )
   END_RUNG wire#w1
   RUNG wire#powerrail
      Contact( #DATA_VALVE_4.SWITCH_ON )
   END_RUNG wire#w1
   // the same network as SCL:
   #TIMER_ANY_CYCLE_NOT_DONE(IN := (#DATA_VALVE_1.SWITCH_ON OR #DATA_VALVE_2.SWITCH_ON OR #DATA_VALVE_3.SWITCH_ON OR #DATA_VALVE_4.SWITCH_ON) AND NOT #ALL_LUBRICATION_DONE,   // TON
                           PT := #TIMER_ANY_CYCLE_NOT_DONE.PT);
   #ANY_CYCLE_NOT_DONE := #TIMER_ANY_CYCLE_NOT_DONE.Q;
END_REGION

REGION Network 34: LUBRICATION DONE 1 ALARM
   RUNG wire#powerrail
      Contact( #ANY_CYCLE_NOT_DONE )
      I_Contact( #CYCLE_FINISHED_1 )
      wire#w1
      Contact( #O_BYTE_0.LUBRICATION_DONE_1 )
      wire#w2
      Coil( #LUBRICATION_DONE_1_ALARM )
   END_RUNG
   RUNG wire#powerrail
      Contact( #LUBRICATION_DONE_1_ALARM )
      I_Contact( "DB2120_MPP_ITC_IPC".RESET_FAULTS )
   END_RUNG wire#w1
   RUNG wire#w2
      Coil( "DB426_ALARMS_WARNINGS".SERVICES."708803" )
   END_RUNG
   // the same network as SCL:
   #LUBRICATION_DONE_1_ALARM := ((#ANY_CYCLE_NOT_DONE AND NOT #CYCLE_FINISHED_1) OR (#LUBRICATION_DONE_1_ALARM AND NOT "DB2120_MPP_ITC_IPC".RESET_FAULTS)) AND #O_BYTE_0.LUBRICATION_DONE_1;
   "DB426_ALARMS_WARNINGS".SERVICES."708803" := #LUBRICATION_DONE_1_ALARM;
END_REGION

REGION Network 35: LUBRICATION DONE 2 ALARM
   RUNG wire#powerrail
      Contact( #ANY_CYCLE_NOT_DONE )
      I_Contact( #CYCLE_FINISHED_2 )
      wire#w1
      Contact( #O_BYTE_1.LUBRICATION_DONE_2 )
      wire#w2
      Coil( #LUBRICATION_DONE_2_ALARM )
   END_RUNG
   RUNG wire#powerrail
      Contact( #LUBRICATION_DONE_2_ALARM )
      I_Contact( "DB2120_MPP_ITC_IPC".RESET_FAULTS )
   END_RUNG wire#w1
   RUNG wire#w2
      Coil( "DB426_ALARMS_WARNINGS".SERVICES."708804" )
   END_RUNG
   // the same network as SCL:
   #LUBRICATION_DONE_2_ALARM := ((#ANY_CYCLE_NOT_DONE AND NOT #CYCLE_FINISHED_2) OR (#LUBRICATION_DONE_2_ALARM AND NOT "DB2120_MPP_ITC_IPC".RESET_FAULTS)) AND #O_BYTE_1.LUBRICATION_DONE_2;
   "DB426_ALARMS_WARNINGS".SERVICES."708804" := #LUBRICATION_DONE_2_ALARM;
END_REGION

REGION Network 36: LUBRICATION DONE 3 ALARM
   RUNG wire#powerrail
      Contact( #ANY_CYCLE_NOT_DONE )
      I_Contact( #CYCLE_FINISHED_3 )
      wire#w1
      Contact( #O_BYTE_1.LUBRICATION_DONE_3 )
      wire#w2
      Coil( #LUBRICATION_DONE_3_ALARM )
   END_RUNG
   RUNG wire#powerrail
      Contact( #LUBRICATION_DONE_3_ALARM )
      I_Contact( "DB2120_MPP_ITC_IPC".RESET_FAULTS )
   END_RUNG wire#w1
   RUNG wire#w2
      Coil( "DB426_ALARMS_WARNINGS".SERVICES."708805" )
   END_RUNG
   // the same network as SCL:
   #LUBRICATION_DONE_3_ALARM := ((#ANY_CYCLE_NOT_DONE AND NOT #CYCLE_FINISHED_3) OR (#LUBRICATION_DONE_3_ALARM AND NOT "DB2120_MPP_ITC_IPC".RESET_FAULTS)) AND #O_BYTE_1.LUBRICATION_DONE_3;
   "DB426_ALARMS_WARNINGS".SERVICES."708805" := #LUBRICATION_DONE_3_ALARM;
END_REGION

REGION Network 37: LUBRICATION DONE 4 ALARM
   RUNG wire#powerrail
      Contact( #ANY_CYCLE_NOT_DONE )
      I_Contact( #CYCLE_FINISHED_4 )
      wire#w1
      Contact( #O_BYTE_1.LUBRICATION_DONE_4 )
      wire#w2
      Coil( #LUBRICATION_DONE_4_ALARM )
   END_RUNG
   RUNG wire#powerrail
      Contact( #LUBRICATION_DONE_4_ALARM )
      I_Contact( "DB2120_MPP_ITC_IPC".RESET_FAULTS )
   END_RUNG wire#w1
   RUNG wire#w2
      Coil( "DB426_ALARMS_WARNINGS".SERVICES."708806" )
   END_RUNG
   // the same network as SCL:
   #LUBRICATION_DONE_4_ALARM := ((#ANY_CYCLE_NOT_DONE AND NOT #CYCLE_FINISHED_4) OR (#LUBRICATION_DONE_4_ALARM AND NOT "DB2120_MPP_ITC_IPC".RESET_FAULTS)) AND #O_BYTE_1.LUBRICATION_DONE_4;
   "DB426_ALARMS_WARNINGS".SERVICES."708806" := #LUBRICATION_DONE_4_ALARM;
END_REGION

REGION Network 38: STOP END OF CYCLE ALARMS
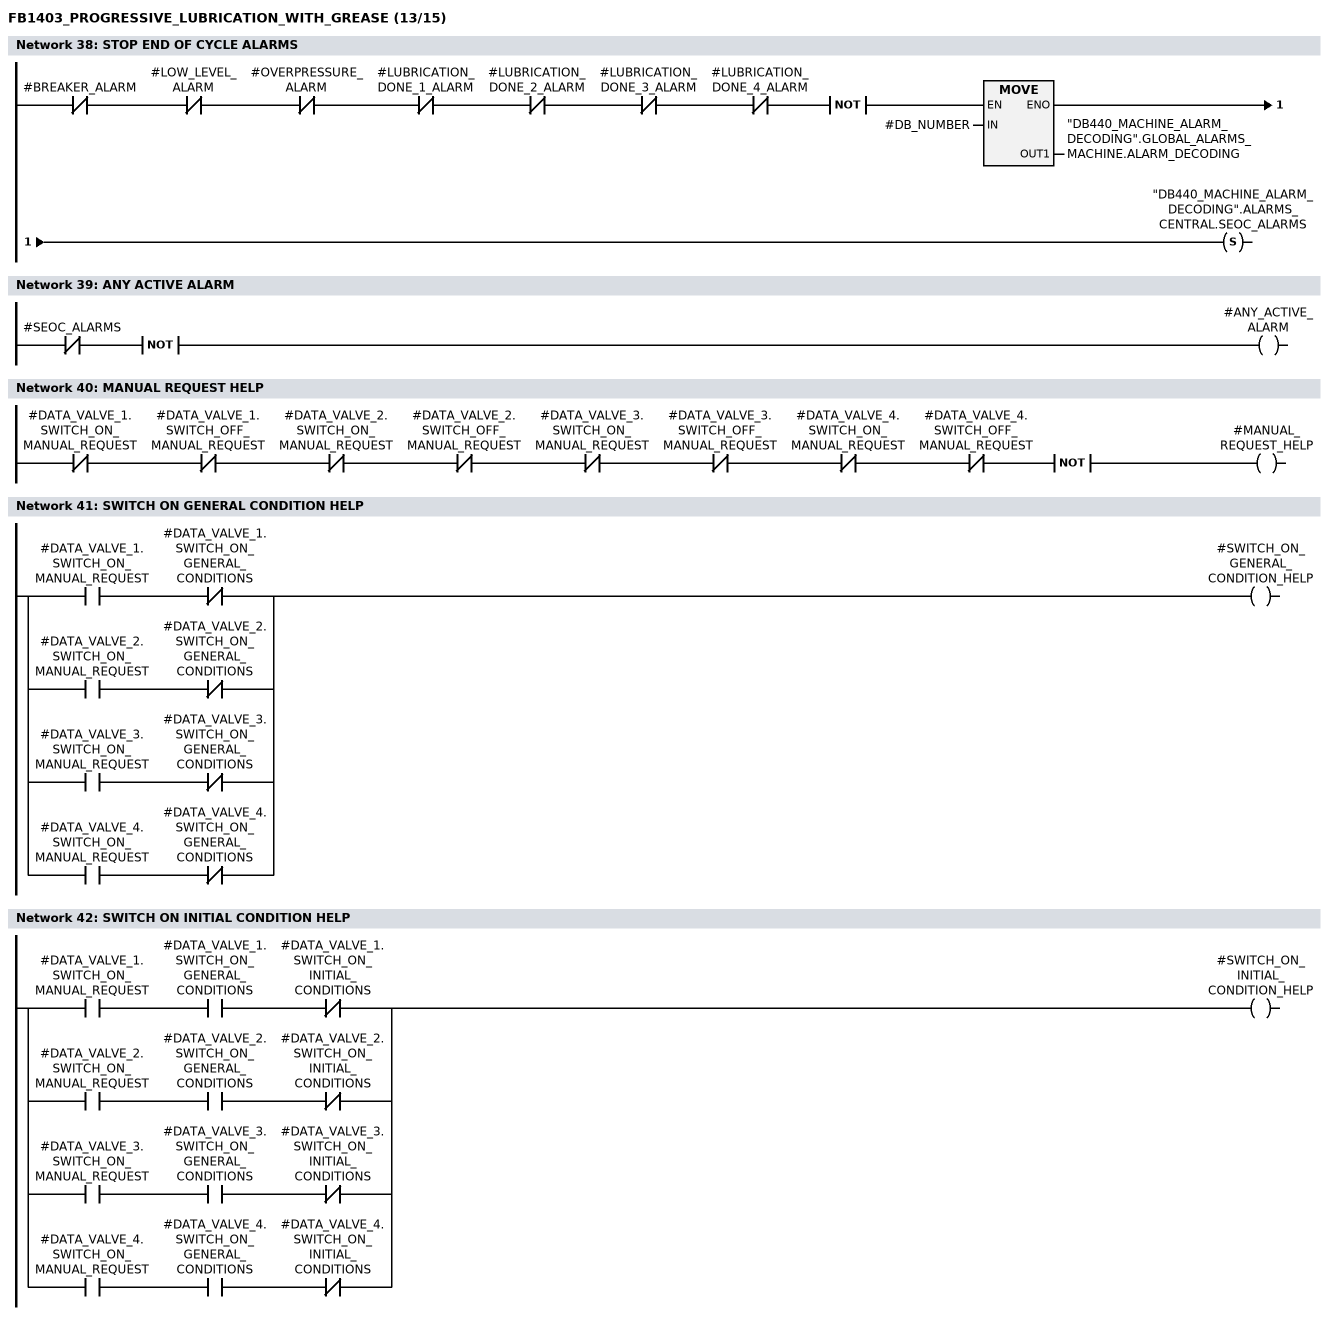
   RUNG wire#powerrail
      I_Contact( #BREAKER_ALARM )
      I_Contact( #LOW_LEVEL_ALARM )
      I_Contact( #OVERPRESSURE_ALARM )
      I_Contact( #LUBRICATION_DONE_1_ALARM )
      I_Contact( #LUBRICATION_DONE_2_ALARM )
      I_Contact( #LUBRICATION_DONE_3_ALARM )
      I_Contact( #LUBRICATION_DONE_4_ALARM )
      Not()
      Move(in := #DB_NUMBER, out1 => "DB440_MACHINE_ALARM_DECODING".GLOBAL_ALARMS_MACHINE.ALARM_DECODING)
      S_Coil( "DB440_MACHINE_ALARM_DECODING".ALARMS_CENTRAL.SEOC_ALARMS )
   END_RUNG
   // the same network as SCL:
   IF NOT (NOT #BREAKER_ALARM AND NOT #LOW_LEVEL_ALARM AND NOT #OVERPRESSURE_ALARM AND NOT #LUBRICATION_DONE_1_ALARM AND NOT #LUBRICATION_DONE_2_ALARM AND NOT #LUBRICATION_DONE_3_ALARM AND NOT #LUBRICATION_DONE_4_ALARM) THEN
       "DB440_MACHINE_ALARM_DECODING".GLOBAL_ALARMS_MACHINE.ALARM_DECODING := #DB_NUMBER;
       "DB440_MACHINE_ALARM_DECODING".ALARMS_CENTRAL.SEOC_ALARMS := TRUE;
   END_IF;
END_REGION

REGION Network 39: ANY ACTIVE ALARM
   RUNG wire#powerrail
      I_Contact( #SEOC_ALARMS )
      Not()
      Coil( #ANY_ACTIVE_ALARM )
   END_RUNG
   // the same network as SCL:
   #ANY_ACTIVE_ALARM := NOT (NOT #SEOC_ALARMS);
END_REGION

REGION Network 40: MANUAL REQUEST HELP
   RUNG wire#powerrail
      I_Contact( #DATA_VALVE_1.SWITCH_ON_MANUAL_REQUEST )
      I_Contact( #DATA_VALVE_1.SWITCH_OFF_MANUAL_REQUEST )
      I_Contact( #DATA_VALVE_2.SWITCH_ON_MANUAL_REQUEST )
      I_Contact( #DATA_VALVE_2.SWITCH_OFF_MANUAL_REQUEST )
      I_Contact( #DATA_VALVE_3.SWITCH_ON_MANUAL_REQUEST )
      I_Contact( #DATA_VALVE_3.SWITCH_OFF_MANUAL_REQUEST )
      I_Contact( #DATA_VALVE_4.SWITCH_ON_MANUAL_REQUEST )
      I_Contact( #DATA_VALVE_4.SWITCH_OFF_MANUAL_REQUEST )
      Not()
      Coil( #MANUAL_REQUEST_HELP )
   END_RUNG
   // the same network as SCL:
   #MANUAL_REQUEST_HELP := NOT (NOT #DATA_VALVE_1.SWITCH_ON_MANUAL_REQUEST AND NOT #DATA_VALVE_1.SWITCH_OFF_MANUAL_REQUEST AND NOT #DATA_VALVE_2.SWITCH_ON_MANUAL_REQUEST AND NOT #DATA_VALVE_2.SWITCH_OFF_MANUAL_REQUEST AND NOT #DATA_VALVE_3.SWITCH_ON_MANUAL_REQUEST AND NOT #DATA_VALVE_3.SWITCH_OFF_MANUAL_REQUEST AND NOT #DATA_VALVE_4.SWITCH_ON_MANUAL_REQUEST AND NOT #DATA_VALVE_4.SWITCH_OFF_MANUAL_REQUEST);
END_REGION

REGION Network 41: SWITCH ON GENERAL CONDITION HELP
   RUNG wire#powerrail
      Contact( #DATA_VALVE_1.SWITCH_ON_MANUAL_REQUEST )
      I_Contact( #DATA_VALVE_1.SWITCH_ON_GENERAL_CONDITIONS )
      wire#w1
      Coil( #SWITCH_ON_GENERAL_CONDITION_HELP )
   END_RUNG
   RUNG wire#powerrail
      Contact( #DATA_VALVE_2.SWITCH_ON_MANUAL_REQUEST )
      I_Contact( #DATA_VALVE_2.SWITCH_ON_GENERAL_CONDITIONS )
   END_RUNG wire#w1
   RUNG wire#powerrail
      Contact( #DATA_VALVE_3.SWITCH_ON_MANUAL_REQUEST )
      I_Contact( #DATA_VALVE_3.SWITCH_ON_GENERAL_CONDITIONS )
   END_RUNG wire#w1
   RUNG wire#powerrail
      Contact( #DATA_VALVE_4.SWITCH_ON_MANUAL_REQUEST )
      I_Contact( #DATA_VALVE_4.SWITCH_ON_GENERAL_CONDITIONS )
   END_RUNG wire#w1
   // the same network as SCL:
   #SWITCH_ON_GENERAL_CONDITION_HELP := (#DATA_VALVE_1.SWITCH_ON_MANUAL_REQUEST AND NOT #DATA_VALVE_1.SWITCH_ON_GENERAL_CONDITIONS) OR (#DATA_VALVE_2.SWITCH_ON_MANUAL_REQUEST AND NOT #DATA_VALVE_2.SWITCH_ON_GENERAL_CONDITIONS) OR (#DATA_VALVE_3.SWITCH_ON_MANUAL_REQUEST AND NOT #DATA_VALVE_3.SWITCH_ON_GENERAL_CONDITIONS) OR (#DATA_VALVE_4.SWITCH_ON_MANUAL_REQUEST AND NOT #DATA_VALVE_4.SWITCH_ON_GENERAL_CONDITIONS);
END_REGION

REGION Network 42: SWITCH ON INITIAL CONDITION HELP
   RUNG wire#powerrail
      Contact( #DATA_VALVE_1.SWITCH_ON_MANUAL_REQUEST )
      Contact( #DATA_VALVE_1.SWITCH_ON_GENERAL_CONDITIONS )
      I_Contact( #DATA_VALVE_1.SWITCH_ON_INITIAL_CONDITIONS )
      wire#w1
      Coil( #SWITCH_ON_INITIAL_CONDITION_HELP )
   END_RUNG
   RUNG wire#powerrail
      Contact( #DATA_VALVE_2.SWITCH_ON_MANUAL_REQUEST )
      Contact( #DATA_VALVE_2.SWITCH_ON_GENERAL_CONDITIONS )
      I_Contact( #DATA_VALVE_2.SWITCH_ON_INITIAL_CONDITIONS )
   END_RUNG wire#w1
   RUNG wire#powerrail
      Contact( #DATA_VALVE_3.SWITCH_ON_MANUAL_REQUEST )
      Contact( #DATA_VALVE_3.SWITCH_ON_GENERAL_CONDITIONS )
      I_Contact( #DATA_VALVE_3.SWITCH_ON_INITIAL_CONDITIONS )
   END_RUNG wire#w1
   RUNG wire#powerrail
      Contact( #DATA_VALVE_4.SWITCH_ON_MANUAL_REQUEST )
      Contact( #DATA_VALVE_4.SWITCH_ON_GENERAL_CONDITIONS )
      I_Contact( #DATA_VALVE_4.SWITCH_ON_INITIAL_CONDITIONS )
   END_RUNG wire#w1
   // the same network as SCL:
   #SWITCH_ON_INITIAL_CONDITION_HELP := (#DATA_VALVE_1.SWITCH_ON_MANUAL_REQUEST AND #DATA_VALVE_1.SWITCH_ON_GENERAL_CONDITIONS AND NOT #DATA_VALVE_1.SWITCH_ON_INITIAL_CONDITIONS) OR (#DATA_VALVE_2.SWITCH_ON_MANUAL_REQUEST AND #DATA_VALVE_2.SWITCH_ON_GENERAL_CONDITIONS AND NOT #DATA_VALVE_2.SWITCH_ON_INITIAL_CONDITIONS) OR (#DATA_VALVE_3.SWITCH_ON_MANUAL_REQUEST AND #DATA_VALVE_3.SWITCH_ON_GENERAL_CONDITIONS AND NOT #DATA_VALVE_3.SWITCH_ON_INITIAL_CONDITIONS) OR (#DATA_VALVE_4.SWITCH_ON_MANUAL_REQUEST AND #DATA_VALVE_4.SWITCH_ON_GENERAL_CONDITIONS AND NOT #DATA_VALVE_4.SWITCH_ON_INITIAL_CONDITIONS);
END_REGION

REGION Network 43: SWITCH OFF GENERAL CONDITION HELP
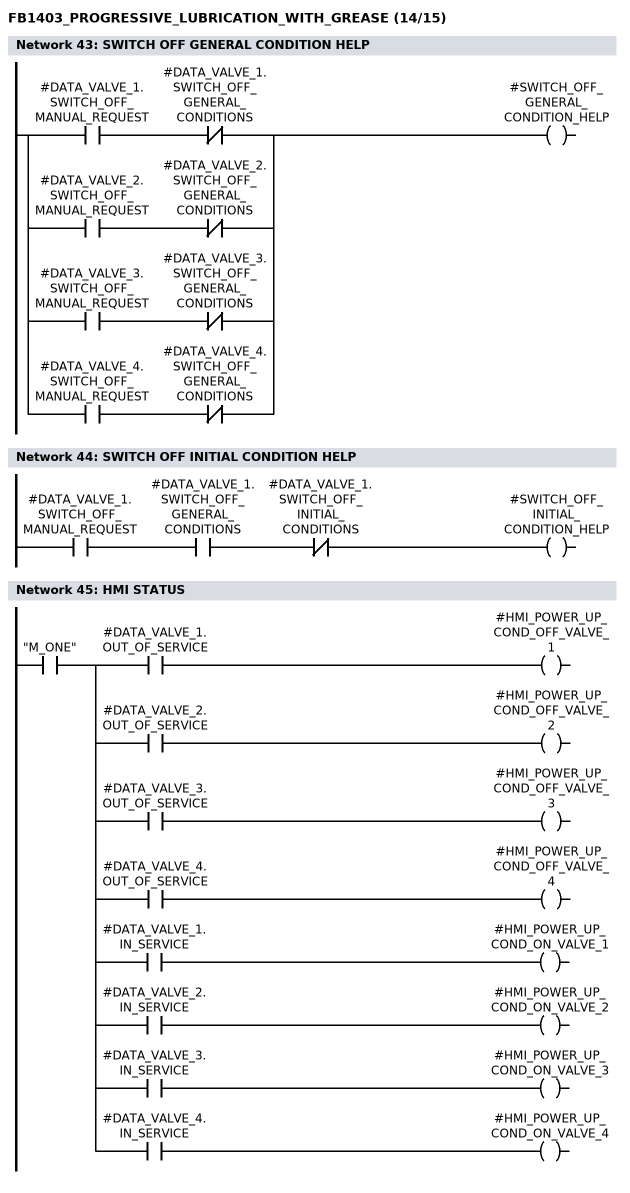
   RUNG wire#powerrail
      Contact( #DATA_VALVE_1.SWITCH_OFF_MANUAL_REQUEST )
      I_Contact( #DATA_VALVE_1.SWITCH_OFF_GENERAL_CONDITIONS )
      wire#w1
      Coil( #SWITCH_OFF_GENERAL_CONDITION_HELP )
   END_RUNG
   RUNG wire#powerrail
      Contact( #DATA_VALVE_2.SWITCH_OFF_MANUAL_REQUEST )
      I_Contact( #DATA_VALVE_2.SWITCH_OFF_GENERAL_CONDITIONS )
   END_RUNG wire#w1
   RUNG wire#powerrail
      Contact( #DATA_VALVE_3.SWITCH_OFF_MANUAL_REQUEST )
      I_Contact( #DATA_VALVE_3.SWITCH_OFF_GENERAL_CONDITIONS )
   END_RUNG wire#w1
   RUNG wire#powerrail
      Contact( #DATA_VALVE_4.SWITCH_OFF_MANUAL_REQUEST )
      I_Contact( #DATA_VALVE_4.SWITCH_OFF_GENERAL_CONDITIONS )
   END_RUNG wire#w1
   // the same network as SCL:
   #SWITCH_OFF_GENERAL_CONDITION_HELP := (#DATA_VALVE_1.SWITCH_OFF_MANUAL_REQUEST AND NOT #DATA_VALVE_1.SWITCH_OFF_GENERAL_CONDITIONS) OR (#DATA_VALVE_2.SWITCH_OFF_MANUAL_REQUEST AND NOT #DATA_VALVE_2.SWITCH_OFF_GENERAL_CONDITIONS) OR (#DATA_VALVE_3.SWITCH_OFF_MANUAL_REQUEST AND NOT #DATA_VALVE_3.SWITCH_OFF_GENERAL_CONDITIONS) OR (#DATA_VALVE_4.SWITCH_OFF_MANUAL_REQUEST AND NOT #DATA_VALVE_4.SWITCH_OFF_GENERAL_CONDITIONS);
END_REGION

REGION Network 44: SWITCH OFF INITIAL CONDITION HELP
   RUNG wire#powerrail
      Contact( #DATA_VALVE_1.SWITCH_OFF_MANUAL_REQUEST )
      Contact( #DATA_VALVE_1.SWITCH_OFF_GENERAL_CONDITIONS )
      I_Contact( #DATA_VALVE_1.SWITCH_OFF_INITIAL_CONDITIONS )
      Coil( #SWITCH_OFF_INITIAL_CONDITION_HELP )
   END_RUNG
   // the same network as SCL:
   #SWITCH_OFF_INITIAL_CONDITION_HELP := #DATA_VALVE_1.SWITCH_OFF_MANUAL_REQUEST AND #DATA_VALVE_1.SWITCH_OFF_GENERAL_CONDITIONS AND NOT #DATA_VALVE_1.SWITCH_OFF_INITIAL_CONDITIONS;
END_REGION

REGION Network 45: HMI STATUS
   RUNG wire#powerrail
      Contact( "M_ONE" )
      wire#w1
      Contact( #DATA_VALVE_1.OUT_OF_SERVICE )
      Coil( #HMI_POWER_UP_COND_OFF_VALVE_1 )
   END_RUNG
   RUNG wire#w1
      Contact( #DATA_VALVE_2.OUT_OF_SERVICE )
      Coil( #HMI_POWER_UP_COND_OFF_VALVE_2 )
   END_RUNG
   RUNG wire#w1
      Contact( #DATA_VALVE_3.OUT_OF_SERVICE )
      Coil( #HMI_POWER_UP_COND_OFF_VALVE_3 )
   END_RUNG
   RUNG wire#w1
      Contact( #DATA_VALVE_4.OUT_OF_SERVICE )
      Coil( #HMI_POWER_UP_COND_OFF_VALVE_4 )
   END_RUNG
   RUNG wire#w1
      Contact( #DATA_VALVE_1.IN_SERVICE )
      Coil( #HMI_POWER_UP_COND_ON_VALVE_1 )
   END_RUNG
   RUNG wire#w1
      Contact( #DATA_VALVE_2.IN_SERVICE )
      Coil( #HMI_POWER_UP_COND_ON_VALVE_2 )
   END_RUNG
   RUNG wire#w1
      Contact( #DATA_VALVE_3.IN_SERVICE )
      Coil( #HMI_POWER_UP_COND_ON_VALVE_3 )
   END_RUNG
   RUNG wire#w1
      Contact( #DATA_VALVE_4.IN_SERVICE )
      Coil( #HMI_POWER_UP_COND_ON_VALVE_4 )
   END_RUNG
   // the same network as SCL:
   #HMI_POWER_UP_COND_OFF_VALVE_1 := "M_ONE" AND #DATA_VALVE_1.OUT_OF_SERVICE;
   #HMI_POWER_UP_COND_OFF_VALVE_2 := "M_ONE" AND #DATA_VALVE_2.OUT_OF_SERVICE;
   #HMI_POWER_UP_COND_OFF_VALVE_3 := "M_ONE" AND #DATA_VALVE_3.OUT_OF_SERVICE;
   #HMI_POWER_UP_COND_OFF_VALVE_4 := "M_ONE" AND #DATA_VALVE_4.OUT_OF_SERVICE;
   #HMI_POWER_UP_COND_ON_VALVE_1 := "M_ONE" AND #DATA_VALVE_1.IN_SERVICE;
   #HMI_POWER_UP_COND_ON_VALVE_2 := "M_ONE" AND #DATA_VALVE_2.IN_SERVICE;
   #HMI_POWER_UP_COND_ON_VALVE_3 := "M_ONE" AND #DATA_VALVE_3.IN_SERVICE;
   #HMI_POWER_UP_COND_ON_VALVE_4 := "M_ONE" AND #DATA_VALVE_4.IN_SERVICE;
END_REGION

REGION Network 46: HMI STATUS
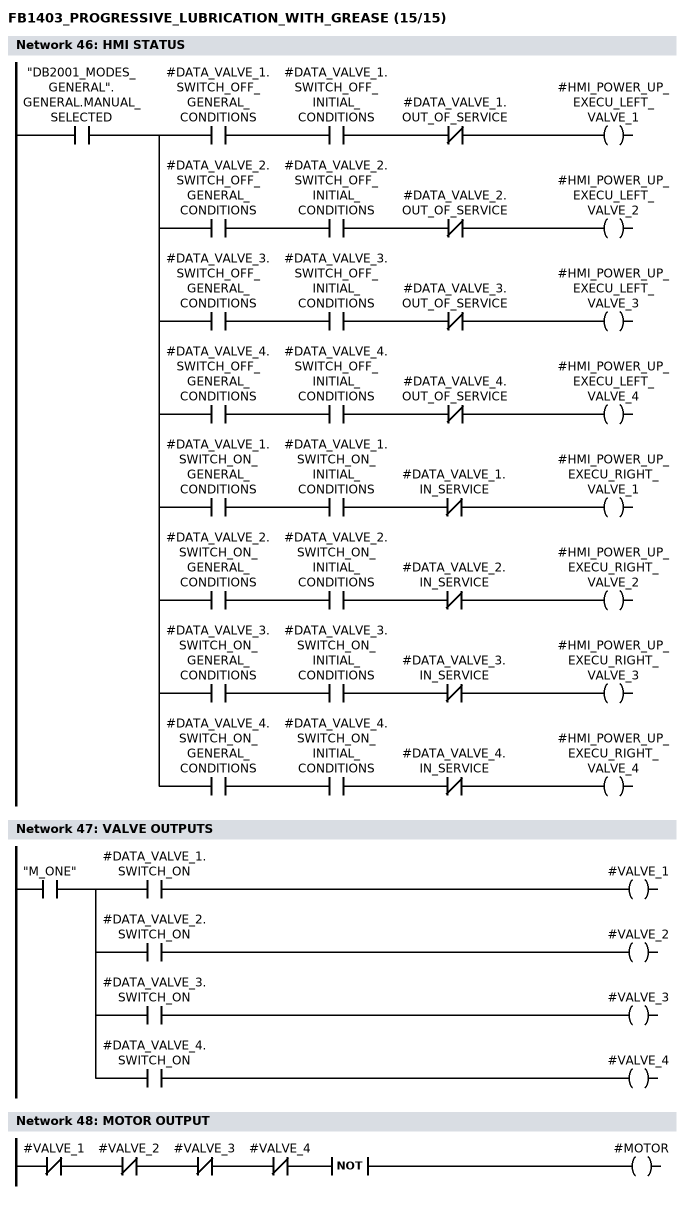
   RUNG wire#powerrail
      Contact( "DB2001_MODES_GENERAL".GENERAL.MANUAL_SELECTED )
      wire#w1
      Contact( #DATA_VALVE_1.SWITCH_OFF_GENERAL_CONDITIONS )
      Contact( #DATA_VALVE_1.SWITCH_OFF_INITIAL_CONDITIONS )
      I_Contact( #DATA_VALVE_1.OUT_OF_SERVICE )
      Coil( #HMI_POWER_UP_EXECU_LEFT_VALVE_1 )
   END_RUNG
   RUNG wire#w1
      Contact( #DATA_VALVE_2.SWITCH_OFF_GENERAL_CONDITIONS )
      Contact( #DATA_VALVE_2.SWITCH_OFF_INITIAL_CONDITIONS )
      I_Contact( #DATA_VALVE_2.OUT_OF_SERVICE )
      Coil( #HMI_POWER_UP_EXECU_LEFT_VALVE_2 )
   END_RUNG
   RUNG wire#w1
      Contact( #DATA_VALVE_3.SWITCH_OFF_GENERAL_CONDITIONS )
      Contact( #DATA_VALVE_3.SWITCH_OFF_INITIAL_CONDITIONS )
      I_Contact( #DATA_VALVE_3.OUT_OF_SERVICE )
      Coil( #HMI_POWER_UP_EXECU_LEFT_VALVE_3 )
   END_RUNG
   RUNG wire#w1
      Contact( #DATA_VALVE_4.SWITCH_OFF_GENERAL_CONDITIONS )
      Contact( #DATA_VALVE_4.SWITCH_OFF_INITIAL_CONDITIONS )
      I_Contact( #DATA_VALVE_4.OUT_OF_SERVICE )
      Coil( #HMI_POWER_UP_EXECU_LEFT_VALVE_4 )
   END_RUNG
   RUNG wire#w1
      Contact( #DATA_VALVE_1.SWITCH_ON_GENERAL_CONDITIONS )
      Contact( #DATA_VALVE_1.SWITCH_ON_INITIAL_CONDITIONS )
      I_Contact( #DATA_VALVE_1.IN_SERVICE )
      Coil( #HMI_POWER_UP_EXECU_RIGHT_VALVE_1 )
   END_RUNG
   RUNG wire#w1
      Contact( #DATA_VALVE_2.SWITCH_ON_GENERAL_CONDITIONS )
      Contact( #DATA_VALVE_2.SWITCH_ON_INITIAL_CONDITIONS )
      I_Contact( #DATA_VALVE_2.IN_SERVICE )
      Coil( #HMI_POWER_UP_EXECU_RIGHT_VALVE_2 )
   END_RUNG
   RUNG wire#w1
      Contact( #DATA_VALVE_3.SWITCH_ON_GENERAL_CONDITIONS )
      Contact( #DATA_VALVE_3.SWITCH_ON_INITIAL_CONDITIONS )
      I_Contact( #DATA_VALVE_3.IN_SERVICE )
      Coil( #HMI_POWER_UP_EXECU_RIGHT_VALVE_3 )
   END_RUNG
   RUNG wire#w1
      Contact( #DATA_VALVE_4.SWITCH_ON_GENERAL_CONDITIONS )
      Contact( #DATA_VALVE_4.SWITCH_ON_INITIAL_CONDITIONS )
      I_Contact( #DATA_VALVE_4.IN_SERVICE )
      Coil( #HMI_POWER_UP_EXECU_RIGHT_VALVE_4 )
   END_RUNG
   // the same network as SCL:
   #HMI_POWER_UP_EXECU_LEFT_VALVE_1 := "DB2001_MODES_GENERAL".GENERAL.MANUAL_SELECTED AND #DATA_VALVE_1.SWITCH_OFF_GENERAL_CONDITIONS AND #DATA_VALVE_1.SWITCH_OFF_INITIAL_CONDITIONS AND NOT #DATA_VALVE_1.OUT_OF_SERVICE;
   #HMI_POWER_UP_EXECU_LEFT_VALVE_2 := "DB2001_MODES_GENERAL".GENERAL.MANUAL_SELECTED AND #DATA_VALVE_2.SWITCH_OFF_GENERAL_CONDITIONS AND #DATA_VALVE_2.SWITCH_OFF_INITIAL_CONDITIONS AND NOT #DATA_VALVE_2.OUT_OF_SERVICE;
   #HMI_POWER_UP_EXECU_LEFT_VALVE_3 := "DB2001_MODES_GENERAL".GENERAL.MANUAL_SELECTED AND #DATA_VALVE_3.SWITCH_OFF_GENERAL_CONDITIONS AND #DATA_VALVE_3.SWITCH_OFF_INITIAL_CONDITIONS AND NOT #DATA_VALVE_3.OUT_OF_SERVICE;
   #HMI_POWER_UP_EXECU_LEFT_VALVE_4 := "DB2001_MODES_GENERAL".GENERAL.MANUAL_SELECTED AND #DATA_VALVE_4.SWITCH_OFF_GENERAL_CONDITIONS AND #DATA_VALVE_4.SWITCH_OFF_INITIAL_CONDITIONS AND NOT #DATA_VALVE_4.OUT_OF_SERVICE;
   #HMI_POWER_UP_EXECU_RIGHT_VALVE_1 := "DB2001_MODES_GENERAL".GENERAL.MANUAL_SELECTED AND #DATA_VALVE_1.SWITCH_ON_GENERAL_CONDITIONS AND #DATA_VALVE_1.SWITCH_ON_INITIAL_CONDITIONS AND NOT #DATA_VALVE_1.IN_SERVICE;
   #HMI_POWER_UP_EXECU_RIGHT_VALVE_2 := "DB2001_MODES_GENERAL".GENERAL.MANUAL_SELECTED AND #DATA_VALVE_2.SWITCH_ON_GENERAL_CONDITIONS AND #DATA_VALVE_2.SWITCH_ON_INITIAL_CONDITIONS AND NOT #DATA_VALVE_2.IN_SERVICE;
   #HMI_POWER_UP_EXECU_RIGHT_VALVE_3 := "DB2001_MODES_GENERAL".GENERAL.MANUAL_SELECTED AND #DATA_VALVE_3.SWITCH_ON_GENERAL_CONDITIONS AND #DATA_VALVE_3.SWITCH_ON_INITIAL_CONDITIONS AND NOT #DATA_VALVE_3.IN_SERVICE;
   #HMI_POWER_UP_EXECU_RIGHT_VALVE_4 := "DB2001_MODES_GENERAL".GENERAL.MANUAL_SELECTED AND #DATA_VALVE_4.SWITCH_ON_GENERAL_CONDITIONS AND #DATA_VALVE_4.SWITCH_ON_INITIAL_CONDITIONS AND NOT #DATA_VALVE_4.IN_SERVICE;
END_REGION

REGION Network 47: VALVE OUTPUTS
   RUNG wire#powerrail
      Contact( "M_ONE" )
      wire#w1
      Contact( #DATA_VALVE_1.SWITCH_ON )
      Coil( #VALVE_1 )
   END_RUNG
   RUNG wire#w1
      Contact( #DATA_VALVE_2.SWITCH_ON )
      Coil( #VALVE_2 )
   END_RUNG
   RUNG wire#w1
      Contact( #DATA_VALVE_3.SWITCH_ON )
      Coil( #VALVE_3 )
   END_RUNG
   RUNG wire#w1
      Contact( #DATA_VALVE_4.SWITCH_ON )
      Coil( #VALVE_4 )
   END_RUNG
   // the same network as SCL:
   #VALVE_1 := "M_ONE" AND #DATA_VALVE_1.SWITCH_ON;
   #VALVE_2 := "M_ONE" AND #DATA_VALVE_2.SWITCH_ON;
   #VALVE_3 := "M_ONE" AND #DATA_VALVE_3.SWITCH_ON;
   #VALVE_4 := "M_ONE" AND #DATA_VALVE_4.SWITCH_ON;
END_REGION

REGION Network 48: MOTOR OUTPUT
   RUNG wire#powerrail
      I_Contact( #VALVE_1 )
      I_Contact( #VALVE_2 )
      I_Contact( #VALVE_3 )
      I_Contact( #VALVE_4 )
      Not()
      Coil( #MOTOR )
   END_RUNG
   // the same network as SCL:
   #MOTOR := NOT (NOT #VALVE_1 AND NOT #VALVE_2 AND NOT #VALVE_3 AND NOT #VALVE_4);
END_REGION
END_FUNCTION_BLOCK
